LIN {X 0,Y 264.267,Z 962.971,A -85,B 0,C 180,E1 -27558.932,E2 -27558.932} C_VEL
LIN {X 0,Y 248.377,Z 979.382,A -85,B 0,C 180,E1 -27561.576,E2 -27561.576} C_VEL
LIN {X 0,Y 232.266,Z 994.174,A -85,B 0,C 180,E1 -27564.723,E2 -27564.723} C_VEL
LIN {X 0,Y 216.727,Z 1007.351,A -85,B 0,C 180,E1 -27568.372,E2 -27568.372} C_VEL
LIN {X 0,Y 201.146,Z 1019.293,A -85,B 0,C 180,E1 -27572.85,E2 -27572.85} C_VEL
LIN {X 0,Y 187.229,Z 1029.33,A -85,B 0,C 180,E1 -27577.891,E2 -27577.891} C_VEL
LIN {X 0,Y 173.48,Z 1038.583,A -85,B 0,C 180,E1 -27584.382,E2 -27584.382} C_VEL
LIN {X 0,Y 162.777,Z 1045.623,A -85,B 0,C 180,E1 -27591.272,E2 -27591.272} C_VEL
LIN {X 0,Y 153.415,Z 1051.791,A -85,B 0,C 180,E1 -27600.094,E2 -27600.094} C_VEL
LIN {X 0,Y 148.288,Z 1055.438,A -85,B 0,C 180,E1 -27607.815,E2 -27607.815} C_VEL
LIN {X 0,Y 145.02,Z 1058.302,A -85,B 0,C 180,E1 -27617.254,E2 -27617.254} C_VEL
LIN {X 0,Y 144.131,Z 1059.404,A -85,B 0,C 180,E1 -27625.225,E2 -27625.225} C_VEL
LIN {X 0,Y 144.059,Z 1059.565,A -85,B 0,C 180,E1 -27631.989,E2 -27631.989} C_VEL
LIN {X 0,Y 144.452,Z 1058.916,A -85,B 0,C 180,E1 -27639.161,E2 -27639.161} C_VEL
LIN {X 0,Y 146.018,Z 1057.309,A -85,B 0,C 180,E1 -27646.715,E2 -27646.715} C_VEL
LIN {X 0,Y 149.982,Z 1054.279,A -85,B 0,C 180,E1 -27655.257,E2 -27655.257} C_VEL
LIN {X 0,Y 157.615,Z 1049.051,A -85,B 0,C 180,E1 -27664.441,E2 -27664.441} C_VEL
LIN {X 0,Y 166.845,Z 1043.052,A -85,B 0,C 180,E1 -27671.699,E2 -27671.699} C_VEL
LIN {X 0,Y 180.107,Z 1034.277,A -85,B 0,C 180,E1 -27679.073,E2 -27679.073} C_VEL
LIN {X 0,Y 192.349,Z 1025.823,A -85,B 0,C 180,E1 -27684.188,E2 -27684.188} C_VEL
LIN {X 0,Y 208.78,Z 1013.706,A -85,B 0,C 180,E1 -27689.548,E2 -27689.548} C_VEL
LIN {X 0,Y 222.856,Z 1002.432,A -85,B 0,C 180,E1 -27693.234,E2 -27693.234} C_VEL
LIN {X 0,Y 239.33,Z 988.118,A -85,B 0,C 180,E1 -27696.8,E2 -27696.8} C_VEL
LIN {X 0,Y 254.068,Z 973.895,A -85,B 0,C 180,E1 -27699.497,E2 -27699.497} C_VEL
LIN {X 0,Y 269.736,Z 957.383,A -85,B 0,C 180,E1 -27701.958,E2 -27701.958} C_VEL
LIN {X 0,Y 284.481,Z 939.789,A -85,B 0,C 180,E1 -27703.988,E2 -27703.988} C_VEL
LIN {X 0,Y 298.698,Z 921.024,A -85,B 0,C 180,E1 -27705.72,E2 -27705.72} C_VEL
LIN {X 0,Y 311.756,Z 901.235,A -85,B 0,C 180,E1 -27707.166,E2 -27707.166} C_VEL
LIN {X 0,Y 323.633,Z 881.021,A -85,B 0,C 180,E1 -27708.35,E2 -27708.35} C_VEL
LIN {X 0,Y 334.691,Z 859.013,A -85,B 0,C 180,E1 -27709.386,E2 -27709.386} C_VEL
LIN {X 0,Y 343.522,Z 838.703,A -85,B 0,C 180,E1 -27710.155,E2 -27710.155} C_VEL
LIN {X 0,Y 352.143,Z 814.942,A -85,B 0,C 180,E1 -27710.876,E2 -27710.876} C_VEL
LIN {X 0,Y 358.427,Z 793.654,A -85,B 0,C 180,E1 -27711.389,E2 -27711.389} C_VEL
LIN {X 0,Y 364.35,Z 767.82,A -85,B 0,C 180,E1 -27711.861,E2 -27711.861} C_VEL
LIN {X 0,Y 367.939,Z 745.502,A -85,B 0,C 180,E1 -27712.18,E2 -27712.18} C_VEL
LIN {X 0,Y 380.155,Z 638.893,A -85,B 0,C 180,E1 -27713.582,E2 -27713.582} C_VEL
LIN {X 0,Y 379.242,Z 636.279,A -85,B 0,C 180,E1 -27715.615,E2 -27715.615} C_VEL
LIN {X 0,Y 378.541,Z 633.63,A -85,B 0,C 180,E1 -27720,E2 -27720} C_VEL
LIN {X 0,Y 379.492,Z 636.936,A -85,B 0,C 180,E1 -27724.685,E2 -27724.685} C_VEL
LIN {X 0,Y 380.192,Z 639.051,A -85,B 0,C 180,E1 -27726.164,E2 -27726.164} C_VEL
LIN {X 0,Y 366.89,Z 754.069,A -85,B 0,C 180,E1 -27727.662,E2 -27727.662} C_VEL
LIN {X 0,Y 362.071,Z 780.264,A -85,B 0,C 180,E1 -27728.054,E2 -27728.054} C_VEL
LIN {X 0,Y 356.568,Z 802.149,A -85,B 0,C 180,E1 -27728.434,E2 -27728.434} C_VEL
LIN {X 0,Y 353.055,Z 813.807,A -85,B 0,C 180,E1 -27728.68,E2 -27728.68} C_VEL
LIN {X 0,Y 350.527,Z 821.162,A -85,B 0,C 180,E1 -27728.649,E2 -27728.649} C_VEL
LIN {X 0,Y 342.323,Z 840.671,A -85,B 0,C 180,E1 -27728.173,E2 -27728.173} C_VEL
LIN {X 0,Y 339.699,Z 846.579,A -85,B 0,C 180,E1 -27728.225,E2 -27728.225} C_VEL
LIN {X 0,Y 329.393,Z 869.145,A -85,B 0,C 180,E1 -27729.009,E2 -27729.009} C_VEL
LIN {X 0,Y 318.229,Z 889.834,A -85,B 0,C 180,E1 -27729.926,E2 -27729.926} C_VEL
LIN {X 0,Y 305.654,Z 910.454,A -85,B 0,C 180,E1 -27731.069,E2 -27731.069} C_VEL
LIN {X 0,Y 291.612,Z 930.378,A -85,B 0,C 180,E1 -27732.475,E2 -27732.475} C_VEL
LIN {X 0,Y 277.331,Z 948.589,A -85,B 0,C 180,E1 -27734.104,E2 -27734.104} C_VEL
LIN {X 0,Y 261.326,Z 966.611,A -85,B 0,C 180,E1 -27736.181,E2 -27736.181} C_VEL
LIN {X 0,Y 246.138,Z 982.117,A -85,B 0,C 180,E1 -27738.473,E2 -27738.473} C_VEL
LIN {X 0,Y 228.96,Z 997.86,A -85,B 0,C 180,E1 -27741.535,E2 -27741.535} C_VEL
LIN {X 0,Y 213.707,Z 1010.632,A -85,B 0,C 180,E1 -27744.812,E2 -27744.812} C_VEL
LIN {X 0,Y 196.327,Z 1023.93,A -85,B 0,C 180,E1 -27749.436,E2 -27749.436} C_VEL
LIN {X 0,Y 182.4,Z 1033.814,A -85,B 0,C 180,E1 -27754.13,E2 -27754.13} C_VEL
LIN {X 0,Y 166.948,Z 1044.167,A -85,B 0,C 180,E1 -27761.006,E2 -27761.006} C_VEL
LIN {X 0,Y 156.007,Z 1051.247,A -85,B 0,C 180,E1 -27767.703,E2 -27767.703} C_VEL
LIN {X 0,Y 145.908,Z 1057.948,A -85,B 0,C 180,E1 -27776.754,E2 -27776.754} C_VEL
LIN {X 0,Y 139.953,Z 1062.241,A -85,B 0,C 180,E1 -27785.519,E2 -27785.519} C_VEL
LIN {X 0,Y 136.886,Z 1065.116,A -85,B 0,C 180,E1 -27794.319,E2 -27794.319} C_VEL
LIN {X 0,Y 135.998,Z 1066.786,A -85,B 0,C 180,E1 -27803.668,E2 -27803.668} C_VEL
LIN {X 0,Y 136.048,Z 1067.121,A -85,B 0,C 180,E1 -27810.421,E2 -27810.421} C_VEL
LIN {X 0,Y 136.022,Z 1066.636,A -85,B 0,C 180,E1 -27817.603,E2 -27817.603} C_VEL
LIN {X 0,Y 137.072,Z 1064.849,A -85,B 0,C 180,E1 -27826.528,E2 -27826.528} C_VEL
LIN {X 0,Y 140.303,Z 1061.923,A -85,B 0,C 180,E1 -27835.165,E2 -27835.165} C_VEL
LIN {X 0,Y 147.301,Z 1056.96,A -85,B 0,C 180,E1 -27844.778,E2 -27844.778} C_VEL
LIN {X 0,Y 156.952,Z 1050.544,A -85,B 0,C 180,E1 -27852.973,E2 -27852.973} C_VEL
LIN {X 0,Y 169.249,Z 1042.625,A -85,B 0,C 180,E1 -27860.176,E2 -27860.176} C_VEL
LIN {X 0,Y 183.726,Z 1032.758,A -85,B 0,C 180,E1 -27866.373,E2 -27866.373} C_VEL
LIN {X 0,Y 199.243,Z 1021.702,A -85,B 0,C 180,E1 -27871.429,E2 -27871.429} C_VEL
LIN {X 0,Y 215.441,Z 1009.024,A -85,B 0,C 180,E1 -27875.603,E2 -27875.603} C_VEL
LIN {X 0,Y 230.594,Z 996.24,A -85,B 0,C 180,E1 -27878.791,E2 -27878.791} C_VEL
LIN {X 0,Y 247.424,Z 980.57,A -85,B 0,C 180,E1 -27881.746,E2 -27881.746} C_VEL
LIN {X 0,Y 261.312,Z 966.334,A -85,B 0,C 180,E1 -27883.828,E2 -27883.828} C_VEL
LIN {X 0,Y 277.317,Z 948.252,A -85,B 0,C 180,E1 -27885.906,E2 -27885.906} C_VEL
LIN {X 0,Y 291.424,Z 930.233,A -85,B 0,C 180,E1 -27887.517,E2 -27887.517} C_VEL
LIN {X 0,Y 305.178,Z 910.722,A -85,B 0,C 180,E1 -27888.897,E2 -27888.897} C_VEL
LIN {X 0,Y 317.749,Z 890.132,A -85,B 0,C 180,E1 -27890.045,E2 -27890.045} C_VEL
LIN {X 0,Y 328.563,Z 870.14,A -85,B 0,C 180,E1 -27890.939,E2 -27890.939} C_VEL
LIN {X 0,Y 338.982,Z 847.539,A -85,B 0,C 180,E1 -27891.736,E2 -27891.736} C_VEL
LIN {X 0,Y 347.083,Z 826.938,A -85,B 0,C 180,E1 -27892.309,E2 -27892.309} C_VEL
LIN {X 0,Y 355.377,Z 801.149,A -85,B 0,C 180,E1 -27892.854,E2 -27892.854} C_VEL
LIN {X 0,Y 360.895,Z 779.258,A -85,B 0,C 180,E1 -27893.213,E2 -27893.213} C_VEL
LIN {X 0,Y 365.786,Z 752.36,A -85,B 0,C 180,E1 -27893.598,E2 -27893.598} C_VEL
LIN {X 0,Y 378.338,Z 645.252,A -85,B 0,C 180,E1 -27894.959,E2 -27894.959} C_VEL
LIN {X 0,Y 377.845,Z 643.846,A -85,B 0,C 180,E1 -27896.207,E2 -27896.207} C_VEL
LIN {X 0,Y 377.267,Z 641.047,A -85,B 0,C 180,E1 -27900.304,E2 -27900.304} C_VEL
LIN {X 0,Y 378.12,Z 644.537,A -85,B 0,C 180,E1 -27904.93,E2 -27904.93} C_VEL
LIN {X 0,Y 378.282,Z 645.473,A -85,B 0,C 180,E1 -27905.413,E2 -27905.413} C_VEL
LIN {X 0,Y 365.783,Z 751.706,A -85,B 0,C 180,E1 -27906.758,E2 -27906.758} C_VEL
LIN {X 0,Y 360.96,Z 777.648,A -85,B 0,C 180,E1 -27907.144,E2 -27907.144} C_VEL
LIN {X 0,Y 355.511,Z 799.249,A -85,B 0,C 180,E1 -27907.55,E2 -27907.55} C_VEL
LIN {X 0,Y 347.486,Z 824.285,A -85,B 0,C 180,E1 -27908.168,E2 -27908.168} C_VEL
LIN {X 0,Y 339.282,Z 845.216,A -85,B 0,C 180,E1 -27908.831,E2 -27908.831} C_VEL
LIN {X 0,Y 328.693,Z 868.101,A -85,B 0,C 180,E1 -27909.732,E2 -27909.732} C_VEL
LIN {X 0,Y 318.082,Z 887.67,A -85,B 0,C 180,E1 -27910.688,E2 -27910.688} C_VEL
LIN {X 0,Y 305.545,Z 908.098,A -85,B 0,C 180,E1 -27911.911,E2 -27911.911} C_VEL
LIN {X 0,Y 291.891,Z 927.376,A -85,B 0,C 180,E1 -27913.38,E2 -27913.38} C_VEL
LIN {X 0,Y 277.553,Z 945.569,A -85,B 0,C 180,E1 -27915.101,E2 -27915.101} C_VEL
LIN {X 0,Y 262.605,Z 962.274,A -85,B 0,C 180,E1 -27917.119,E2 -27917.119} C_VEL
LIN {X 0,Y 248.018,Z 977.098,A -85,B 0,C 180,E1 -27919.374,E2 -27919.374} C_VEL
LIN {X 0,Y 230.582,Z 993.009,A -85,B 0,C 180,E1 -27922.536,E2 -27922.536} C_VEL
LIN {X 0,Y 216.255,Z 1004.884,A -85,B 0,C 180,E1 -27925.629,E2 -27925.629} C_VEL
LIN {X 0,Y 198.972,Z 1017.992,A -85,B 0,C 180,E1 -27930.192,E2 -27930.192} C_VEL
LIN {X 0,Y 185.069,Z 1027.645,A -85,B 0,C 180,E1 -27934.793,E2 -27934.793} C_VEL
LIN {X 0,Y 170.308,Z 1037.306,A -85,B 0,C 180,E1 -27941.114,E2 -27941.114} C_VEL
LIN {X 0,Y 158.413,Z 1044.613,A -85,B 0,C 180,E1 -27948.006,E2 -27948.006} C_VEL
LIN {X 0,Y 148.285,Z 1050.907,A -85,B 0,C 180,E1 -27956.432,E2 -27956.432} C_VEL
LIN {X 0,Y 141.455,Z 1055.193,A -85,B 0,C 180,E1 -27965.352,E2 -27965.352} C_VEL
LIN {X 0,Y 137.778,Z 1057.908,A -85,B 0,C 180,E1 -27973.992,E2 -27973.992} C_VEL
LIN {X 0,Y 136.239,Z 1059.536,A -85,B 0,C 180,E1 -27983.257,E2 -27983.257} C_VEL
LIN {X 0,Y 136.057,Z 1059.844,A -85,B 0,C 180,E1 -27990.843,E2 -27990.843} C_VEL
LIN {X 0,Y 136.415,Z 1059.26,A -85,B 0,C 180,E1 -27998.855,E2 -27998.855} C_VEL
LIN {X 0,Y 138.135,Z 1057.635,A -85,B 0,C 180,E1 -28007.265,E2 -28007.265} C_VEL
LIN {X 0,Y 142.135,Z 1054.805,A -85,B 0,C 180,E1 -28015.859,E2 -28015.859} C_VEL
LIN {X 0,Y 150.472,Z 1049.553,A -85,B 0,C 180,E1 -28025.787,E2 -28025.787} C_VEL
LIN {X 0,Y 159.802,Z 1043.863,A -85,B 0,C 180,E1 -28033.002,E2 -28033.002} C_VEL
LIN {X 0,Y 173.564,Z 1035.328,A -85,B 0,C 180,E1 -28040.531,E2 -28040.531} C_VEL
LIN {X 0,Y 186.98,Z 1026.493,A -85,B 0,C 180,E1 -28045.984,E2 -28045.984} C_VEL
LIN {X 0,Y 203.26,Z 1015.054,A -85,B 0,C 180,E1 -28051.12,E2 -28051.12} C_VEL
LIN {X 0,Y 218.5,Z 1003.277,A -85,B 0,C 180,E1 -28054.97,E2 -28054.97} C_VEL
LIN {X 0,Y 234.581,Z 989.845,A -85,B 0,C 180,E1 -28058.313,E2 -28058.313} C_VEL
LIN {X 0,Y 250.84,Z 974.588,A -85,B 0,C 180,E1 -28061.163,E2 -28061.163} C_VEL
LIN {X 0,Y 266.01,Z 958.994,A -85,B 0,C 180,E1 -28063.437,E2 -28063.437} C_VEL
LIN {X 0,Y 281.477,Z 941.075,A -85,B 0,C 180,E1 -28065.467,E2 -28065.467} C_VEL
LIN {X 0,Y 294.529,Z 924.26,A -85,B 0,C 180,E1 -28066.99,E2 -28066.99} C_VEL
LIN {X 0,Y 308.68,Z 903.638,A -85,B 0,C 180,E1 -28068.485,E2 -28068.485} C_VEL
LIN {X 0,Y 319.891,Z 885.068,A -85,B 0,C 180,E1 -28069.555,E2 -28069.555} C_VEL
LIN {X 0,Y 331.432,Z 863.224,A -85,B 0,C 180,E1 -28070.582,E2 -28070.582} C_VEL
LIN {X 0,Y 340.824,Z 842.289,A -85,B 0,C 180,E1 -28071.368,E2 -28071.368} C_VEL
LIN {X 0,Y 349.564,Z 819.498,A -85,B 0,C 180,E1 -28072.06,E2 -28072.06} C_VEL
LIN {X 0,Y 356.719,Z 796.023,A -85,B 0,C 180,E1 -28072.615,E2 -28072.615} C_VEL
LIN {X 0,Y 362.622,Z 771.737,A -85,B 0,C 180,E1 -28073.055,E2 -28073.055} C_VEL
LIN {X 0,Y 366.721,Z 747.257,A -85,B 0,C 180,E1 -28073.397,E2 -28073.397} C_VEL
LIN {X 0,Y 378.603,Z 645.5,A -85,B 0,C 180,E1 -28074.696,E2 -28074.696} C_VEL
LIN {X 0,Y 378.146,Z 644.074,A -85,B 0,C 180,E1 -28075.906,E2 -28075.906} C_VEL
LIN {X 0,Y 377.562,Z 641.607,A -85,B 0,C 180,E1 -28080,E2 -28080} C_VEL
LIN {X 0,Y 378.441,Z 644.845,A -85,B 0,C 180,E1 -28084.546,E2 -28084.546} C_VEL
LIN {X 0,Y 378.613,Z 645.771,A -85,B 0,C 180,E1 -28085.044,E2 -28085.044} C_VEL
LIN {X 0,Y 365.885,Z 754.02,A -85,B 0,C 180,E1 -28086.417,E2 -28086.417} C_VEL
LIN {X 0,Y 361.033,Z 780.062,A -85,B 0,C 180,E1 -28086.792,E2 -28086.792} C_VEL
LIN {X 0,Y 355.448,Z 802.054,A -85,B 0,C 180,E1 -28087.154,E2 -28087.154} C_VEL
LIN {X 0,Y 347.573,Z 826.478,A -85,B 0,C 180,E1 -28087.671,E2 -28087.671} C_VEL
LIN {X 0,Y 339.699,Z 846.579,A -85,B 0,C 180,E1 -28088.225,E2 -28088.225} C_VEL
LIN {X 0,Y 336.5,Z 853.766,A -85,B 0,C 180,E1 -28088.278,E2 -28088.278} C_VEL
LIN {X 0,Y 327.075,Z 871.41,A -85,B 0,C 180,E1 -28087.878,E2 -28087.878} C_VEL
LIN {X 0,Y 323.395,Z 878.079,A -85,B 0,C 180,E1 -28087.97,E2 -28087.97} C_VEL
LIN {X 0,Y 309.842,Z 901.381,A -85,B 0,C 180,E1 -28089.071,E2 -28089.071} C_VEL
LIN {X 0,Y 297.638,Z 919.683,A -85,B 0,C 180,E1 -28090.162,E2 -28090.162} C_VEL
LIN {X 0,Y 281.872,Z 940.552,A -85,B 0,C 180,E1 -28091.745,E2 -28091.745} C_VEL
LIN {X 0,Y 268.172,Z 956.644,A -85,B 0,C 180,E1 -28093.307,E2 -28093.307} C_VEL
LIN {X 0,Y 252.011,Z 973.807,A -85,B 0,C 180,E1 -28095.417,E2 -28095.417} C_VEL
LIN {X 0,Y 236.296,Z 988.661,A -85,B 0,C 180,E1 -28097.807,E2 -28097.807} C_VEL
LIN {X 0,Y 219.884,Z 1002.877,A -85,B 0,C 180,E1 -28100.775,E2 -28100.775} C_VEL
LIN {X 0,Y 202.401,Z 1016.446,A -85,B 0,C 180,E1 -28104.634,E2 -28104.634} C_VEL
LIN {X 0,Y 186.443,Z 1027.891,A -85,B 0,C 180,E1 -28109.053,E2 -28109.053} C_VEL
LIN {X 0,Y 170.442,Z 1038.405,A -85,B 0,C 180,E1 -28114.784,E2 -28114.784} C_VEL
LIN {X 0,Y 157.522,Z 1046.472,A -85,B 0,C 180,E1 -28120.942,E2 -28120.942} C_VEL
LIN {X 0,Y 144.759,Z 1054.201,A -85,B 0,C 180,E1 -28129.512,E2 -28129.512} C_VEL
LIN {X 0,Y 136.669,Z 1059.222,A -85,B 0,C 180,E1 -28137.718,E2 -28137.718} C_VEL
LIN {X 0,Y 130.717,Z 1063.469,A -85,B 0,C 180,E1 -28147.987,E2 -28147.987} C_VEL
LIN {X 0,Y 128.303,Z 1065.79,A -85,B 0,C 180,E1 -28157.853,E2 -28157.853} C_VEL
LIN {X 0,Y 128.002,Z 1066.673,A -85,B 0,C 180,E1 -28165.07,E2 -28165.07} C_VEL
LIN {X 0,Y 128.037,Z 1066.847,A -85,B 0,C 180,E1 -28171.611,E2 -28171.611} C_VEL
LIN {X 0,Y 128.061,Z 1066.277,A -85,B 0,C 180,E1 -28178.984,E2 -28178.984} C_VEL
LIN {X 0,Y 129.395,Z 1064.512,A -85,B 0,C 180,E1 -28188.004,E2 -28188.004} C_VEL
LIN {X 0,Y 133.243,Z 1061.482,A -85,B 0,C 180,E1 -28197.242,E2 -28197.242} C_VEL
LIN {X 0,Y 141.776,Z 1055.963,A -85,B 0,C 180,E1 -28207.848,E2 -28207.848} C_VEL
LIN {X 0,Y 152.078,Z 1049.679,A -85,B 0,C 180,E1 -28215.818,E2 -28215.818} C_VEL
LIN {X 0,Y 166.561,Z 1040.767,A -85,B 0,C 180,E1 -28223.554,E2 -28223.554} C_VEL
LIN {X 0,Y 180.674,Z 1031.602,A -85,B 0,C 180,E1 -28229.07,E2 -28229.07} C_VEL
LIN {X 0,Y 197.714,Z 1019.773,A -85,B 0,C 180,E1 -28234.182,E2 -28234.182} C_VEL
LIN {X 0,Y 213.604,Z 1007.659,A -85,B 0,C 180,E1 -28237.948,E2 -28237.948} C_VEL
LIN {X 0,Y 231.168,Z 993.076,A -85,B 0,C 180,E1 -28241.332,E2 -28241.332} C_VEL
LIN {X 0,Y 246.727,Z 978.641,A -85,B 0,C 180,E1 -28243.835,E2 -28243.835} C_VEL
LIN {X 0,Y 262.742,Z 962.378,A -85,B 0,C 180,E1 -28246.03,E2 -28246.03} C_VEL
LIN {X 0,Y 278.183,Z 944.676,A -85,B 0,C 180,E1 -28247.867,E2 -28247.867} C_VEL
LIN {X 0,Y 291.565,Z 927.644,A -85,B 0,C 180,E1 -28249.27,E2 -28249.27} C_VEL
LIN {X 0,Y 306.532,Z 906.072,A -85,B 0,C 180,E1 -28250.657,E2 -28250.657} C_VEL
LIN {X 0,Y 317.663,Z 887.817,A -85,B 0,C 180,E1 -28251.592,E2 -28251.592} C_VEL
LIN {X 0,Y 329.774,Z 865.097,A -85,B 0,C 180,E1 -28252.513,E2 -28252.513} C_VEL
LIN {X 0,Y 339.026,Z 844.701,A -85,B 0,C 180,E1 -28253.163,E2 -28253.163} C_VEL
LIN {X 0,Y 348.03,Z 821.467,A -85,B 0,C 180,E1 -28253.749,E2 -28253.749} C_VEL
LIN {X 0,Y 355.282,Z 797.991,A -85,B 0,C 180,E1 -28254.193,E2 -28254.193} C_VEL
LIN {X 0,Y 361.272,Z 773.573,A -85,B 0,C 180,E1 -28254.563,E2 -28254.563} C_VEL
LIN {X 0,Y 365.395,Z 749.119,A -85,B 0,C 180,E1 -28254.89,E2 -28254.89} C_VEL
LIN {X 0,Y 376.897,Z 651.874,A -85,B 0,C 180,E1 -28256.121,E2 -28256.121} C_VEL
LIN {X 0,Y 376.286,Z 649.042,A -85,B 0,C 180,E1 -28260.305,E2 -28260.305} C_VEL
LIN {X 0,Y 376.874,Z 651.979,A -85,B 0,C 180,E1 -28264.279,E2 -28264.279} C_VEL
LIN {X 0,Y 364.904,Z 752.116,A -85,B 0,C 180,E1 -28265.512,E2 -28265.512} C_VEL
LIN {X 0,Y 360.049,Z 777.886,A -85,B 0,C 180,E1 -28265.88,E2 -28265.88} C_VEL
LIN {X 0,Y 354.531,Z 799.534,A -85,B 0,C 180,E1 -28266.268,E2 -28266.268} C_VEL
LIN {X 0,Y 346.437,Z 824.507,A -85,B 0,C 180,E1 -28266.854,E2 -28266.854} C_VEL
LIN {X 0,Y 338.312,Z 845.035,A -85,B 0,C 180,E1 -28267.472,E2 -28267.472} C_VEL
LIN {X 0,Y 327.901,Z 867.426,A -85,B 0,C 180,E1 -28268.304,E2 -28268.304} C_VEL
LIN {X 0,Y 317.061,Z 887.243,A -85,B 0,C 180,E1 -28269.22,E2 -28269.22} C_VEL
LIN {X 0,Y 304.443,Z 907.627,A -85,B 0,C 180,E1 -28270.374,E2 -28270.374} C_VEL
LIN {X 0,Y 290.581,Z 926.992,A -85,B 0,C 180,E1 -28271.773,E2 -28271.773} C_VEL
LIN {X 0,Y 276.451,Z 944.688,A -85,B 0,C 180,E1 -28273.36,E2 -28273.36} C_VEL
LIN {X 0,Y 260.324,Z 962.495,A -85,B 0,C 180,E1 -28275.405,E2 -28275.405} C_VEL
LIN {X 0,Y 245.431,Z 977.318,A -85,B 0,C 180,E1 -28277.576,E2 -28277.576} C_VEL
LIN {X 0,Y 227.57,Z 993.23,A -85,B 0,C 180,E1 -28280.631,E2 -28280.631} C_VEL
LIN {X 0,Y 212.836,Z 1005.105,A -85,B 0,C 180,E1 -28283.638,E2 -28283.638} C_VEL
LIN {X 0,Y 194.97,Z 1018.213,A -85,B 0,C 180,E1 -28288.105,E2 -28288.105} C_VEL
LIN {X 0,Y 180.504,Z 1027.866,A -85,B 0,C 180,E1 -28292.649,E2 -28292.649} C_VEL
LIN {X 0,Y 165.431,Z 1037.293,A -85,B 0,C 180,E1 -28298.768,E2 -28298.768} C_VEL
LIN {X 0,Y 152.41,Z 1044.833,A -85,B 0,C 180,E1 -28305.94,E2 -28305.94} C_VEL
LIN {X 0,Y 141.535,Z 1051.126,A -85,B 0,C 180,E1 -28314.599,E2 -28314.599} C_VEL
LIN {X 0,Y 133.837,Z 1055.565,A -85,B 0,C 180,E1 -28324.322,E2 -28324.322} C_VEL
LIN {X 0,Y 129.755,Z 1058.344,A -85,B 0,C 180,E1 -28333.894,E2 -28333.894} C_VEL
LIN {X 0,Y 128.208,Z 1059.791,A -85,B 0,C 180,E1 -28343.732,E2 -28343.732} C_VEL
LIN {X 0,Y 128.062,Z 1060.035,A -85,B 0,C 180,E1 -28351.343,E2 -28351.343} C_VEL
LIN {X 0,Y 128.471,Z 1059.475,A -85,B 0,C 180,E1 -28359.407,E2 -28359.407} C_VEL
LIN {X 0,Y 130.413,Z 1057.851,A -85,B 0,C 180,E1 -28368.322,E2 -28368.322} C_VEL
LIN {X 0,Y 134.841,Z 1055.022,A -85,B 0,C 180,E1 -28377.371,E2 -28377.371} C_VEL
LIN {X 0,Y 143.899,Z 1049.771,A -85,B 0,C 180,E1 -28387.696,E2 -28387.696} C_VEL
LIN {X 0,Y 153.895,Z 1044.081,A -85,B 0,C 180,E1 -28395.089,E2 -28395.089} C_VEL
LIN {X 0,Y 167.826,Z 1035.944,A -85,B 0,C 180,E1 -28402.411,E2 -28402.411} C_VEL
LIN {X 0,Y 181.805,Z 1027.162,A -85,B 0,C 180,E1 -28407.884,E2 -28407.884} C_VEL
LIN {X 0,Y 197.9,Z 1016.396,A -85,B 0,C 180,E1 -28412.779,E2 -28412.779} C_VEL
LIN {X 0,Y 214.351,Z 1004.121,A -85,B 0,C 180,E1 -28416.774,E2 -28416.774} C_VEL
LIN {X 0,Y 230.838,Z 990.757,A -85,B 0,C 180,E1 -28420.044,E2 -28420.044} C_VEL
LIN {X 0,Y 247.08,Z 976,A -85,B 0,C 180,E1 -28422.756,E2 -28422.756} C_VEL
LIN {X 0,Y 261.13,Z 961.963,A -85,B 0,C 180,E1 -28424.781,E2 -28424.781} C_VEL
LIN {X 0,Y 278.07,Z 943.085,A -85,B 0,C 180,E1 -28426.907,E2 -28426.907} C_VEL
LIN {X 0,Y 291.429,Z 926.286,A -85,B 0,C 180,E1 -28428.392,E2 -28428.392} C_VEL
LIN {X 0,Y 305.772,Z 906.042,A -85,B 0,C 180,E1 -28429.83,E2 -28429.83} C_VEL
LIN {X 0,Y 317.471,Z 887.094,A -85,B 0,C 180,E1 -28430.89,E2 -28430.89} C_VEL
LIN {X 0,Y 328.953,Z 866.044,A -85,B 0,C 180,E1 -28431.855,E2 -28431.855} C_VEL
LIN {X 0,Y 338.758,Z 844.749,A -85,B 0,C 180,E1 -28432.635,E2 -28432.635} C_VEL
LIN {X 0,Y 346.867,Z 824.239,A -85,B 0,C 180,E1 -28433.249,E2 -28433.249} C_VEL
LIN {X 0,Y 355.048,Z 798.859,A -85,B 0,C 180,E1 -28433.842,E2 -28433.842} C_VEL
LIN {X 0,Y 360.569,Z 777.071,A -85,B 0,C 180,E1 -28434.23,E2 -28434.23} C_VEL
LIN {X 0,Y 365.485,Z 750.335,A -85,B 0,C 180,E1 -28434.606,E2 -28434.606} C_VEL
LIN {X 0,Y 377.199,Z 652.091,A -85,B 0,C 180,E1 -28435.819,E2 -28435.819} C_VEL
LIN {X 0,Y 376.582,Z 649.582,A -85,B 0,C 180,E1 -28440,E2 -28440} C_VEL
LIN {X 0,Y 377.201,Z 652.309,A -85,B 0,C 180,E1 -28443.913,E2 -28443.913} C_VEL
LIN {X 0,Y 365.076,Z 753.823,A -85,B 0,C 180,E1 -28445.165,E2 -28445.165} C_VEL
LIN {X 0,Y 360.144,Z 779.979,A -85,B 0,C 180,E1 -28445.525,E2 -28445.525} C_VEL
LIN {X 0,Y 354.506,Z 801.959,A -85,B 0,C 180,E1 -28445.867,E2 -28445.867} C_VEL
LIN {X 0,Y 346.59,Z 826.271,A -85,B 0,C 180,E1 -28446.351,E2 -28446.351} C_VEL
LIN {X 0,Y 338.24,Z 847.311,A -85,B 0,C 180,E1 -28446.901,E2 -28446.901} C_VEL
LIN {X 0,Y 327.875,Z 869.594,A -85,B 0,C 180,E1 -28447.64,E2 -28447.64} C_VEL
LIN {X 0,Y 323.395,Z 878.079,A -85,B 0,C 180,E1 -28447.97,E2 -28447.97} C_VEL
LIN {X 0,Y 319.555,Z 884.853,A -85,B 0,C 180,E1 -28448.078,E2 -28448.078} C_VEL
LIN {X 0,Y 308.524,Z 901.631,A -85,B 0,C 180,E1 -28447.786,E2 -28447.786} C_VEL
LIN {X 0,Y 304.263,Z 907.989,A -85,B 0,C 180,E1 -28447.938,E2 -28447.938} C_VEL
LIN {X 0,Y 289.417,Z 928.793,A -85,B 0,C 180,E1 -28449.227,E2 -28449.227} C_VEL
LIN {X 0,Y 275.661,Z 945.924,A -85,B 0,C 180,E1 -28450.584,E2 -28450.584} C_VEL
LIN {X 0,Y 258.148,Z 965.245,A -85,B 0,C 180,E1 -28452.557,E2 -28452.557} C_VEL
LIN {X 0,Y 243.077,Z 980.109,A -85,B 0,C 180,E1 -28454.532,E2 -28454.532} C_VEL
LIN {X 0,Y 224.294,Z 996.716,A -85,B 0,C 180,E1 -28457.446,E2 -28457.446} C_VEL
LIN {X 0,Y 208.975,Z 1008.909,A -85,B 0,C 180,E1 -28460.313,E2 -28460.313} C_VEL
LIN {X 0,Y 191.086,Z 1021.923,A -85,B 0,C 180,E1 -28464.427,E2 -28464.427} C_VEL
LIN {X 0,Y 175.092,Z 1032.441,A -85,B 0,C 180,E1 -28469.105,E2 -28469.105} C_VEL
LIN {X 0,Y 159.14,Z 1042.284,A -85,B 0,C 180,E1 -28475.234,E2 -28475.234} C_VEL
LIN {X 0,Y 145.278,Z 1050.186,A -85,B 0,C 180,E1 -28482.571,E2 -28482.571} C_VEL
LIN {X 0,Y 133.636,Z 1056.854,A -85,B 0,C 180,E1 -28491.609,E2 -28491.609} C_VEL
LIN {X 0,Y 125.456,Z 1061.638,A -85,B 0,C 180,E1 -28501.95,E2 -28501.95} C_VEL
LIN {X 0,Y 121.399,Z 1064.563,A -85,B 0,C 180,E1 -28511.761,E2 -28511.761} C_VEL
LIN {X 0,Y 120.022,Z 1066.338,A -85,B 0,C 180,E1 -28522.472,E2 -28522.472} C_VEL
LIN {X 0,Y 120.061,Z 1066.713,A -85,B 0,C 180,E1 -28530,E2 -28530} C_VEL
LIN {X 0,Y 120.026,Z 1066.324,A -85,B 0,C 180,E1 -28537.659,E2 -28537.659} C_VEL
LIN {X 0,Y 121.399,Z 1064.531,A -85,B 0,C 180,E1 -28548.239,E2 -28548.239} C_VEL
LIN {X 0,Y 125.452,Z 1061.594,A -85,B 0,C 180,E1 -28558.05,E2 -28558.05} C_VEL
LIN {X 0,Y 133.632,Z 1056.786,A -85,B 0,C 180,E1 -28568.392,E2 -28568.392} C_VEL
LIN {X 0,Y 145.272,Z 1050.1,A -85,B 0,C 180,E1 -28577.431,E2 -28577.431} C_VEL
LIN {X 0,Y 159.132,Z 1042.18,A -85,B 0,C 180,E1 -28584.769,E2 -28584.769} C_VEL
LIN {X 0,Y 175.084,Z 1032.312,A -85,B 0,C 180,E1 -28590.899,E2 -28590.899} C_VEL
LIN {X 0,Y 191.867,Z 1021.256,A -85,B 0,C 180,E1 -28595.781,E2 -28595.781} C_VEL
LIN {X 0,Y 208.964,Z 1008.723,A -85,B 0,C 180,E1 -28599.694,E2 -28599.694} C_VEL
LIN {X 0,Y 225.151,Z 995.796,A -85,B 0,C 180,E1 -28602.709,E2 -28602.709} C_VEL
LIN {X 0,Y 242.94,Z 979.967,A -85,B 0,C 180,E1 -28605.459,E2 -28605.459} C_VEL
LIN {X 0,Y 258.137,Z 964.957,A -85,B 0,C 180,E1 -28607.452,E2 -28607.452} C_VEL
LIN {X 0,Y 275.65,Z 945.572,A -85,B 0,C 180,E1 -28609.426,E2 -28609.426} C_VEL
LIN {X 0,Y 289.23,Z 928.628,A -85,B 0,C 180,E1 -28610.767,E2 -28610.767} C_VEL
LIN {X 0,Y 304.104,Z 907.734,A -85,B 0,C 180,E1 -28612.062,E2 -28612.062} C_VEL
LIN {X 0,Y 315.827,Z 888.874,A -85,B 0,C 180,E1 -28612.988,E2 -28612.988} C_VEL
LIN {X 0,Y 327.372,Z 867.881,A -85,B 0,C 180,E1 -28613.809,E2 -28613.809} C_VEL
LIN {X 0,Y 337.527,Z 845.96,A -85,B 0,C 180,E1 -28614.481,E2 -28614.481} C_VEL
LIN {X 0,Y 345.784,Z 825.204,A -85,B 0,C 180,E1 -28614.986,E2 -28614.986} C_VEL
LIN {X 0,Y 353.859,Z 800.264,A -85,B 0,C 180,E1 -28615.446,E2 -28615.446} C_VEL
LIN {X 0,Y 359.472,Z 778.283,A -85,B 0,C 180,E1 -28615.765,E2 -28615.765} C_VEL
LIN {X 0,Y 364.36,Z 751.781,A -85,B 0,C 180,E1 -28616.112,E2 -28616.112} C_VEL
LIN {X 0,Y 375.552,Z 659.084,A -85,B 0,C 180,E1 -28617.253,E2 -28617.253} C_VEL
LIN {X 0,Y 375.304,Z 657.034,A -85,B 0,C 180,E1 -28620.305,E2 -28620.305} C_VEL
LIN {X 0,Y 375.524,Z 659.258,A -85,B 0,C 180,E1 -28623.147,E2 -28623.147} C_VEL
LIN {X 0,Y 364.208,Z 752.452,A -85,B 0,C 180,E1 -28624.26,E2 -28624.26} C_VEL
LIN {X 0,Y 359.315,Z 778.125,A -85,B 0,C 180,E1 -28624.61,E2 -28624.61} C_VEL
LIN {X 0,Y 353.728,Z 799.821,A -85,B 0,C 180,E1 -28624.979,E2 -28624.979} C_VEL
LIN {X 0,Y 345.572,Z 824.729,A -85,B 0,C 180,E1 -28625.534,E2 -28625.534} C_VEL
LIN {X 0,Y 337.247,Z 845.523,A -85,B 0,C 180,E1 -28626.127,E2 -28626.127} C_VEL
LIN {X 0,Y 326.357,Z 868.542,A -85,B 0,C 180,E1 -28626.943,E2 -28626.943} C_VEL
LIN {X 0,Y 315.868,Z 887.464,A -85,B 0,C 180,E1 -28627.775,E2 -28627.775} C_VEL
LIN {X 0,Y 303.091,Z 907.847,A -85,B 0,C 180,E1 -28628.87,E2 -28628.87} C_VEL
LIN {X 0,Y 289.036,Z 927.212,A -85,B 0,C 180,E1 -28630.2,E2 -28630.2} C_VEL
LIN {X 0,Y 274.688,Z 944.908,A -85,B 0,C 180,E1 -28631.711,E2 -28631.711} C_VEL
LIN {X 0,Y 258.28,Z 962.715,A -85,B 0,C 180,E1 -28633.663,E2 -28633.663} C_VEL
LIN {X 0,Y 242.969,Z 977.654,A -85,B 0,C 180,E1 -28635.76,E2 -28635.76} C_VEL
LIN {X 0,Y 224.817,Z 993.451,A -85,B 0,C 180,E1 -28638.679,E2 -28638.679} C_VEL
LIN {X 0,Y 209.683,Z 1005.326,A -85,B 0,C 180,E1 -28641.586,E2 -28641.586} C_VEL
LIN {X 0,Y 191.238,Z 1018.434,A -85,B 0,C 180,E1 -28645.934,E2 -28645.934} C_VEL
LIN {X 0,Y 176.205,Z 1028.087,A -85,B 0,C 180,E1 -28650.398,E2 -28650.398} C_VEL
LIN {X 0,Y 160.412,Z 1037.514,A -85,B 0,C 180,E1 -28656.478,E2 -28656.478} C_VEL
LIN {X 0,Y 146.621,Z 1045.053,A -85,B 0,C 180,E1 -28663.708,E2 -28663.708} C_VEL
LIN {X 0,Y 134.942,Z 1051.345,A -85,B 0,C 180,E1 -28672.584,E2 -28672.584} C_VEL
LIN {X 0,Y 126.541,Z 1055.783,A -85,B 0,C 180,E1 -28682.723,E2 -28682.723} C_VEL
LIN {X 0,Y 121.997,Z 1058.56,A -85,B 0,C 180,E1 -28692.839,E2 -28692.839} C_VEL
LIN {X 0,Y 120.234,Z 1060.005,A -85,B 0,C 180,E1 -28703.314,E2 -28703.314} C_VEL
LIN {X 0,Y 120.065,Z 1060.249,A -85,B 0,C 180,E1 -28711.432,E2 -28711.432} C_VEL
LIN {X 0,Y 120.533,Z 1059.689,A -85,B 0,C 180,E1 -28720.033,E2 -28720.033} C_VEL
LIN {X 0,Y 122.739,Z 1058.067,A -85,B 0,C 180,E1 -28729.513,E2 -28729.513} C_VEL
LIN {X 0,Y 127.65,Z 1055.239,A -85,B 0,C 180,E1 -28739.056,E2 -28739.056} C_VEL
LIN {X 0,Y 137.5,Z 1049.989,A -85,B 0,C 180,E1 -28749.787,E2 -28749.787} C_VEL
LIN {X 0,Y 148.209,Z 1044.3,A -85,B 0,C 180,E1 -28757.339,E2 -28757.339} C_VEL
LIN {X 0,Y 163.604,Z 1035.765,A -85,B 0,C 180,E1 -28764.982,E2 -28764.982} C_VEL
LIN {X 0,Y 178.3,Z 1026.929,A -85,B 0,C 180,E1 -28770.369,E2 -28770.369} C_VEL
LIN {X 0,Y 195.854,Z 1015.489,A -85,B 0,C 180,E1 -28775.332,E2 -28775.332} C_VEL
LIN {X 0,Y 212.253,Z 1003.582,A -85,B 0,C 180,E1 -28779.021,E2 -28779.021} C_VEL
LIN {X 0,Y 229.902,Z 989.529,A -85,B 0,C 180,E1 -28782.265,E2 -28782.265} C_VEL
LIN {X 0,Y 245.672,Z 975.378,A -85,B 0,C 180,E1 -28784.709,E2 -28784.709} C_VEL
LIN {X 0,Y 260.925,Z 960.341,A -85,B 0,C 180,E1 -28786.744,E2 -28786.744} C_VEL
LIN {X 0,Y 277.385,Z 942.053,A -85,B 0,C 180,E1 -28788.661,E2 -28788.661} C_VEL
LIN {X 0,Y 290.841,Z 925.289,A -85,B 0,C 180,E1 -28790.053,E2 -28790.053} C_VEL
LIN {X 0,Y 305.656,Z 904.382,A -85,B 0,C 180,E1 -28791.436,E2 -28791.436} C_VEL
LIN {X 0,Y 317.196,Z 885.77,A -85,B 0,C 180,E1 -28792.408,E2 -28792.408} C_VEL
LIN {X 0,Y 329.18,Z 863.641,A -85,B 0,C 180,E1 -28793.349,E2 -28793.349} C_VEL
LIN {X 0,Y 338.785,Z 842.704,A -85,B 0,C 180,E1 -28794.056,E2 -28794.056} C_VEL
LIN {X 0,Y 347.711,Z 819.908,A -85,B 0,C 180,E1 -28794.679,E2 -28794.679} C_VEL
LIN {X 0,Y 355.029,Z 796.382,A -85,B 0,C 180,E1 -28795.182,E2 -28795.182} C_VEL
LIN {X 0,Y 361.055,Z 772.033,A -85,B 0,C 180,E1 -28795.579,E2 -28795.579} C_VEL
LIN {X 0,Y 365.226,Z 747.641,A -85,B 0,C 180,E1 -28795.893,E2 -28795.893} C_VEL
LIN {X 0,Y 375.855,Z 659.371,A -85,B 0,C 180,E1 -28796.95,E2 -28796.95} C_VEL
LIN {X 0,Y 375.603,Z 657.559,A -85,B 0,C 180,E1 -28800,E2 -28800} C_VEL
LIN {X 0,Y 375.852,Z 659.564,A -85,B 0,C 180,E1 -28802.781,E2 -28802.781} C_VEL
LIN {X 0,Y 364.403,Z 753.898,A -85,B 0,C 180,E1 -28803.91,E2 -28803.91} C_VEL
LIN {X 0,Y 359.455,Z 779.8,A -85,B 0,C 180,E1 -28804.251,E2 -28804.251} C_VEL
LIN {X 0,Y 353.745,Z 801.864,A -85,B 0,C 180,E1 -28804.574,E2 -28804.574} C_VEL
LIN {X 0,Y 345.792,Z 826.065,A -85,B 0,C 180,E1 -28805.026,E2 -28805.026} C_VEL
LIN {X 0,Y 337.535,Z 846.709,A -85,B 0,C 180,E1 -28805.531,E2 -28805.531} C_VEL
LIN {X 0,Y 326.898,Z 869.384,A -85,B 0,C 180,E1 -28806.235,E2 -28806.235} C_VEL
LIN {X 0,Y 315.837,Z 889.411,A -85,B 0,C 180,E1 -28807.025,E2 -28807.025} C_VEL
LIN {X 0,Y 304.263,Z 907.989,A -85,B 0,C 180,E1 -28807.938,E2 -28807.938} C_VEL
LIN {X 0,Y 299.852,Z 914.346,A -85,B 0,C 180,E1 -28808.104,E2 -28808.104} C_VEL
LIN {X 0,Y 287.262,Z 930.021,A -85,B 0,C 180,E1 -28807.921,E2 -28807.921} C_VEL
LIN {X 0,Y 282.464,Z 935.989,A -85,B 0,C 180,E1 -28808.139,E2 -28808.139} C_VEL
LIN {X 0,Y 266.752,Z 954.171,A -85,B 0,C 180,E1 -28809.657,E2 -28809.657} C_VEL
LIN {X 0,Y 251.859,Z 969.696,A -85,B 0,C 180,E1 -28811.303,E2 -28811.303} C_VEL
LIN {X 0,Y 233.588,Z 986.67,A -85,B 0,C 180,E1 -28813.666,E2 -28813.666} C_VEL
LIN {X 0,Y 217.547,Z 1000.039,A -85,B 0,C 180,E1 -28816.135,E2 -28816.135} C_VEL
LIN {X 0,Y 197.755,Z 1014.846,A -85,B 0,C 180,E1 -28819.871,E2 -28819.871} C_VEL
LIN {X 0,Y 181.603,Z 1025.724,A -85,B 0,C 180,E1 -28823.699,E2 -28823.699} C_VEL
LIN {X 0,Y 163.001,Z 1037.139,A -85,B 0,C 180,E1 -28829.417,E2 -28829.417} C_VEL
LIN {X 0,Y 148.479,Z 1045.31,A -85,B 0,C 180,E1 -28835.428,E2 -28835.428} C_VEL
LIN {X 0,Y 134.186,Z 1052.977,A -85,B 0,C 180,E1 -28843.714,E2 -28843.714} C_VEL
LIN {X 0,Y 123.432,Z 1058.569,A -85,B 0,C 180,E1 -28853.169,E2 -28853.169} C_VEL
LIN {X 0,Y 115.915,Z 1062.906,A -85,B 0,C 180,E1 -28864.449,E2 -28864.449} C_VEL
LIN {X 0,Y 112.495,Z 1065.358,A -85,B 0,C 180,E1 -28876.114,E2 -28876.114} C_VEL
LIN {X 0,Y 112.006,Z 1066.269,A -85,B 0,C 180,E1 -28884.878,E2 -28884.878} C_VEL
LIN {X 0,Y 112.04,Z 1066.424,A -85,B 0,C 180,E1 -28891.738,E2 -28891.738} C_VEL
LIN {X 0,Y 112.129,Z 1065.845,A -85,B 0,C 180,E1 -28900.273,E2 -28900.273} C_VEL
LIN {X 0,Y 113.984,Z 1064.075,A -85,B 0,C 180,E1 -28910.541,E2 -28910.541} C_VEL
LIN {X 0,Y 118.9,Z 1061.021,A -85,B 0,C 180,E1 -28920.933,E2 -28920.933} C_VEL
LIN {X 0,Y 129.111,Z 1055.519,A -85,B 0,C 180,E1 -28932.358,E2 -28932.358} C_VEL
LIN {X 0,Y 140.981,Z 1049.257,A -85,B 0,C 180,E1 -28940.63,E2 -28940.63} C_VEL
LIN {X 0,Y 157.27,Z 1040.322,A -85,B 0,C 180,E1 -28948.423,E2 -28948.423} C_VEL
LIN {X 0,Y 172.731,Z 1031.156,A -85,B 0,C 180,E1 -28953.798,E2 -28953.798} C_VEL
LIN {X 0,Y 191.083,Z 1019.327,A -85,B 0,C 180,E1 -28958.658,E2 -28958.658} C_VEL
LIN {X 0,Y 207.961,Z 1007.214,A -85,B 0,C 180,E1 -28962.174,E2 -28962.174} C_VEL
LIN {X 0,Y 226.401,Z 992.655,A -85,B 0,C 180,E1 -28965.285,E2 -28965.285} C_VEL
LIN {X 0,Y 242.663,Z 978.197,A -85,B 0,C 180,E1 -28967.568,E2 -28967.568} C_VEL
LIN {X 0,Y 258.341,Z 962.868,A -85,B 0,C 180,E1 -28969.447,E2 -28969.447} C_VEL
LIN {X 0,Y 274.739,Z 944.791,A -85,B 0,C 180,E1 -28971.151,E2 -28971.151} C_VEL
LIN {X 0,Y 288.497,Z 927.813,A -85,B 0,C 180,E1 -28972.407,E2 -28972.407} C_VEL
LIN {X 0,Y 303.835,Z 906.367,A -85,B 0,C 180,E1 -28973.642,E2 -28973.642} C_VEL
LIN {X 0,Y 315.424,Z 887.837,A -85,B 0,C 180,E1 -28974.487,E2 -28974.487} C_VEL
LIN {X 0,Y 327.359,Z 866.103,A -85,B 0,C 180,E1 -28975.269,E2 -28975.269} C_VEL
LIN {X 0,Y 336.847,Z 845.738,A -85,B 0,C 180,E1 -28975.846,E2 -28975.846} C_VEL
LIN {X 0,Y 345.88,Z 823.129,A -85,B 0,C 180,E1 -28976.354,E2 -28976.354} C_VEL
LIN {X 0,Y 353.607,Z 798.995,A -85,B 0,C 180,E1 -28976.76,E2 -28976.76} C_VEL
LIN {X 0,Y 359.399,Z 776.228,A -85,B 0,C 180,E1 -28977.068,E2 -28977.068} C_VEL
LIN {X 0,Y 364.01,Z 750.794,A -85,B 0,C 180,E1 -28977.383,E2 -28977.383} C_VEL
LIN {X 0,Y 374.357,Z 666.292,A -85,B 0,C 180,E1 -28978.385,E2 -28978.385} C_VEL
LIN {X 0,Y 374.323,Z 665.024,A -85,B 0,C 180,E1 -28980.306,E2 -28980.306} C_VEL
LIN {X 0,Y 374.328,Z 666.477,A -85,B 0,C 180,E1 -28982.006,E2 -28982.006} C_VEL
LIN {X 0,Y 363.684,Z 752.807,A -85,B 0,C 180,E1 -28983.004,E2 -28983.004} C_VEL
LIN {X 0,Y 358.72,Z 778.521,A -85,B 0,C 180,E1 -28983.338,E2 -28983.338} C_VEL
LIN {X 0,Y 353.065,Z 800.251,A -85,B 0,C 180,E1 -28983.687,E2 -28983.687} C_VEL
LIN {X 0,Y 344.89,Z 824.951,A -85,B 0,C 180,E1 -28984.207,E2 -28984.207} C_VEL
LIN {X 0,Y 336.621,Z 845.427,A -85,B 0,C 180,E1 -28984.757,E2 -28984.757} C_VEL
LIN {X 0,Y 325.964,Z 867.867,A -85,B 0,C 180,E1 -28985.501,E2 -28985.501} C_VEL
LIN {X 0,Y 314.878,Z 887.684,A -85,B 0,C 180,E1 -28986.32,E2 -28986.32} C_VEL
LIN {X 0,Y 301.95,Z 908.068,A -85,B 0,C 180,E1 -28987.354,E2 -28987.354} C_VEL
LIN {X 0,Y 287.982,Z 927.086,A -85,B 0,C 180,E1 -28988.586,E2 -28988.586} C_VEL
LIN {X 0,Y 273.674,Z 944.515,A -85,B 0,C 180,E1 -28989.989,E2 -28989.989} C_VEL
LIN {X 0,Y 257.399,Z 962.017,A -85,B 0,C 180,E1 -28991.787,E2 -28991.787} C_VEL
LIN {X 0,Y 242.81,Z 976.085,A -85,B 0,C 180,E1 -28993.629,E2 -28993.629} C_VEL
LIN {X 0,Y 224.92,Z 991.632,A -85,B 0,C 180,E1 -28996.264,E2 -28996.264} C_VEL
LIN {X 0,Y 208.509,Z 1004.292,A -85,B 0,C 180,E1 -28999.145,E2 -28999.145} C_VEL
LIN {X 0,Y 191.027,Z 1016.602,A -85,B 0,C 180,E1 -29002.893,E2 -29002.893} C_VEL
LIN {X 0,Y 173.705,Z 1027.406,A -85,B 0,C 180,E1 -29007.568,E2 -29007.568} C_VEL
LIN {X 0,Y 157.722,Z 1036.602,A -85,B 0,C 180,E1 -29013.194,E2 -29013.194} C_VEL
LIN {X 0,Y 142.25,Z 1044.681,A -85,B 0,C 180,E1 -29020.612,E2 -29020.612} C_VEL
LIN {X 0,Y 130.399,Z 1050.592,A -85,B 0,C 180,E1 -29028.743,E2 -29028.743} C_VEL
LIN {X 0,Y 120.299,Z 1055.539,A -85,B 0,C 180,E1 -29039.535,E2 -29039.535} C_VEL
LIN {X 0,Y 114.96,Z 1058.34,A -85,B 0,C 180,E1 -29049.641,E2 -29049.641} C_VEL
LIN {X 0,Y 112.504,Z 1060.003,A -85,B 0,C 180,E1 -29060.279,E2 -29060.279} C_VEL
LIN {X 0,Y 112.064,Z 1060.497,A -85,B 0,C 180,E1 -29069.489,E2 -29069.489} C_VEL
LIN {X 0,Y 112.386,Z 1060.16,A -85,B 0,C 180,E1 -29078.7,E2 -29078.7} C_VEL
LIN {X 0,Y 114.755,Z 1058.501,A -85,B 0,C 180,E1 -29089.866,E2 -29089.866} C_VEL
LIN {X 0,Y 119.929,Z 1055.765,A -85,B 0,C 180,E1 -29100.016,E2 -29100.016} C_VEL
LIN {X 0,Y 129.86,Z 1050.951,A -85,B 0,C 180,E1 -29110.881,E2 -29110.881} C_VEL
LIN {X 0,Y 141.581,Z 1045.11,A -85,B 0,C 180,E1 -29119.084,E2 -29119.084} C_VEL
LIN {X 0,Y 156.265,Z 1037.543,A -85,B 0,C 180,E1 -29126.287,E2 -29126.287} C_VEL
LIN {X 0,Y 172.862,Z 1028.05,A -85,B 0,C 180,E1 -29132.252,E2 -29132.252} C_VEL
LIN {X 0,Y 190.131,Z 1017.345,A -85,B 0,C 180,E1 -29136.973,E2 -29136.973} C_VEL
LIN {X 0,Y 207.579,Z 1005.182,A -85,B 0,C 180,E1 -29140.755,E2 -29140.755} C_VEL
LIN {X 0,Y 223.135,Z 993.268,A -85,B 0,C 180,E1 -29143.528,E2 -29143.528} C_VEL
LIN {X 0,Y 241.839,Z 977.268,A -85,B 0,C 180,E1 -29146.317,E2 -29146.317} C_VEL
LIN {X 0,Y 256.415,Z 963.31,A -85,B 0,C 180,E1 -29148.175,E2 -29148.175} C_VEL
LIN {X 0,Y 273.098,Z 945.572,A -85,B 0,C 180,E1 -29150.026,E2 -29150.026} C_VEL
LIN {X 0,Y 287.659,Z 927.919,A -85,B 0,C 180,E1 -29151.46,E2 -29151.46} C_VEL
LIN {X 0,Y 301.903,Z 908.627,A -85,B 0,C 180,E1 -29152.717,E2 -29152.717} C_VEL
LIN {X 0,Y 314.837,Z 888.323,A -85,B 0,C 180,E1 -29153.751,E2 -29153.751} C_VEL
LIN {X 0,Y 325.927,Z 868.56,A -85,B 0,C 180,E1 -29154.571,E2 -29154.571} C_VEL
LIN {X 0,Y 336.589,Z 846.29,A -85,B 0,C 180,E1 -29155.313,E2 -29155.313} C_VEL
LIN {X 0,Y 344.861,Z 825.932,A -85,B 0,C 180,E1 -29155.864,E2 -29155.864} C_VEL
LIN {X 0,Y 353.315,Z 800.587,A -85,B 0,C 180,E1 -29156.401,E2 -29156.401} C_VEL
LIN {X 0,Y 359.006,Z 778.773,A -85,B 0,C 180,E1 -29156.752,E2 -29156.752} C_VEL
LIN {X 0,Y 363.948,Z 753.392,A -85,B 0,C 180,E1 -29157.082,E2 -29157.082} C_VEL
LIN {X 0,Y 373.22,Z 678.604,A -85,B 0,C 180,E1 -29157.947,E2 -29157.947} C_VEL
LIN {X 0,Y 374.663,Z 666.562,A -85,B 0,C 180,E1 -29158.123,E2 -29158.123} C_VEL
LIN {X 0,Y 374.623,Z 665.537,A -85,B 0,C 180,E1 -29160,E2 -29160} C_VEL
LIN {X 0,Y 374.642,Z 666.892,A -85,B 0,C 180,E1 -29161.643,E2 -29161.643} C_VEL
LIN {X 0,Y 363.928,Z 753.813,A -85,B 0,C 180,E1 -29162.65,E2 -29162.65} C_VEL
LIN {X 0,Y 358.928,Z 779.688,A -85,B 0,C 180,E1 -29162.974,E2 -29162.974} C_VEL
LIN {X 0,Y 353.164,Z 801.769,A -85,B 0,C 180,E1 -29163.276,E2 -29163.276} C_VEL
LIN {X 0,Y 344.689,Z 827.145,A -85,B 0,C 180,E1 -29163.721,E2 -29163.721} C_VEL
LIN {X 0,Y 336.364,Z 847.634,A -85,B 0,C 180,E1 -29164.194,E2 -29164.194} C_VEL
LIN {X 0,Y 325.145,Z 870.981,A -85,B 0,C 180,E1 -29164.883,E2 -29164.883} C_VEL
LIN {X 0,Y 314.464,Z 890.014,A -85,B 0,C 180,E1 -29165.595,E2 -29165.595} C_VEL
LIN {X 0,Y 301.364,Z 910.636,A -85,B 0,C 180,E1 -29166.563,E2 -29166.563} C_VEL
LIN {X 0,Y 287.075,Z 930.051,A -85,B 0,C 180,E1 -29167.726,E2 -29167.726} C_VEL
LIN {X 0,Y 282.464,Z 935.989,A -85,B 0,C 180,E1 -29168.139,E2 -29168.139} C_VEL
LIN {X 0,Y 277.563,Z 941.904,A -85,B 0,C 180,E1 -29168.379,E2 -29168.379} C_VEL
LIN {X 0,Y 263.612,Z 956.415,A -85,B 0,C 180,E1 -29168.342,E2 -29168.342} C_VEL
LIN {X 0,Y 258.17,Z 961.767,A -85,B 0,C 180,E1 -29168.645,E2 -29168.645} C_VEL
LIN {X 0,Y 241.966,Z 977.394,A -85,B 0,C 180,E1 -29170.422,E2 -29170.422} C_VEL
LIN {X 0,Y 224.458,Z 992.678,A -85,B 0,C 180,E1 -29172.689,E2 -29172.689} C_VEL
LIN {X 0,Y 206.477,Z 1006.544,A -85,B 0,C 180,E1 -29175.488,E2 -29175.488} C_VEL
LIN {X 0,Y 189.941,Z 1018.113,A -85,B 0,C 180,E1 -29178.637,E2 -29178.637} C_VEL
LIN {X 0,Y 170.042,Z 1030.602,A -85,B 0,C 180,E1 -29183.462,E2 -29183.462} C_VEL
LIN {X 0,Y 154.573,Z 1039.395,A -85,B 0,C 180,E1 -29188.388,E2 -29188.388} C_VEL
LIN {X 0,Y 137.157,Z 1048.504,A -85,B 0,C 180,E1 -29195.981,E2 -29195.981} C_VEL
LIN {X 0,Y 124.18,Z 1054.848,A -85,B 0,C 180,E1 -29204.223,E2 -29204.223} C_VEL
LIN {X 0,Y 112.935,Z 1060.369,A -85,B 0,C 180,E1 -29215.484,E2 -29215.484} C_VEL
LIN {X 0,Y 106.753,Z 1063.651,A -85,B 0,C 180,E1 -29226.834,E2 -29226.834} C_VEL
LIN {X 0,Y 104.276,Z 1065.504,A -85,B 0,C 180,E1 -29237.821,E2 -29237.821} C_VEL
LIN {X 0,Y 104.02,Z 1066.154,A -85,B 0,C 180,E1 -29246.693,E2 -29246.693} C_VEL
LIN {X 0,Y 104.027,Z 1066.172,A -85,B 0,C 180,E1 -29252.754,E2 -29252.754} C_VEL
LIN {X 0,Y 104.225,Z 1065.557,A -85,B 0,C 180,E1 -29261.622,E2 -29261.622} C_VEL
LIN {X 0,Y 106.558,Z 1063.738,A -85,B 0,C 180,E1 -29272.626,E2 -29272.626} C_VEL
LIN {X 0,Y 112.571,Z 1060.489,A -85,B 0,C 180,E1 -29284.027,E2 -29284.027} C_VEL
LIN {X 0,Y 123.645,Z 1055.036,A -85,B 0,C 180,E1 -29295.368,E2 -29295.368} C_VEL
LIN {X 0,Y 136.193,Z 1048.877,A -85,B 0,C 180,E1 -29303.51,E2 -29303.51} C_VEL
LIN {X 0,Y 153.824,Z 1039.686,A -85,B 0,C 180,E1 -29311.345,E2 -29311.345} C_VEL
LIN {X 0,Y 170.032,Z 1030.467,A -85,B 0,C 180,E1 -29316.544,E2 -29316.544} C_VEL
LIN {X 0,Y 189.931,Z 1017.942,A -85,B 0,C 180,E1 -29321.37,E2 -29321.37} C_VEL
LIN {X 0,Y 206.467,Z 1006.349,A -85,B 0,C 180,E1 -29324.52,E2 -29324.52} C_VEL
LIN {X 0,Y 225.359,Z 991.654,A -85,B 0,C 180,E1 -29327.45,E2 -29327.45} C_VEL
LIN {X 0,Y 241.957,Z 977.122,A -85,B 0,C 180,E1 -29329.588,E2 -29329.588} C_VEL
LIN {X 0,Y 259.355,Z 960.236,A -85,B 0,C 180,E1 -29331.486,E2 -29331.486} C_VEL
LIN {X 0,Y 275.036,Z 942.893,A -85,B 0,C 180,E1 -29332.97,E2 -29332.97} C_VEL
LIN {X 0,Y 289.467,Z 925.143,A -85,B 0,C 180,E1 -29334.166,E2 -29334.166} C_VEL
LIN {X 0,Y 304.016,Z 904.669,A -85,B 0,C 180,E1 -29335.236,E2 -29335.236} C_VEL
LIN {X 0,Y 316.216,Z 885.171,A -85,B 0,C 180,E1 -29336.049,E2 -29336.049} C_VEL
LIN {X 0,Y 328.48,Z 862.413,A -85,B 0,C 180,E1 -29336.784,E2 -29336.784} C_VEL
LIN {X 0,Y 337.674,Z 842.493,A -85,B 0,C 180,E1 -29337.284,E2 -29337.284} C_VEL
LIN {X 0,Y 347.224,Z 817.83,A -85,B 0,C 180,E1 -29337.77,E2 -29337.77} C_VEL
LIN {X 0,Y 353.968,Z 796.227,A -85,B 0,C 180,E1 -29338.095,E2 -29338.095} C_VEL
LIN {X 0,Y 360.099,Z 771.254,A -85,B 0,C 180,E1 -29338.405,E2 -29338.405} C_VEL
LIN {X 0,Y 364.118,Z 747.875,A -85,B 0,C 180,E1 -29338.678,E2 -29338.678} C_VEL
LIN {X 0,Y 373.312,Z 673.46,A -85,B 0,C 180,E1 -29339.54,E2 -29339.54} C_VEL
LIN {X 0,Y 373.342,Z 673.015,A -85,B 0,C 180,E1 -29340.307,E2 -29340.307} C_VEL
LIN {X 0,Y 373.296,Z 673.577,A -85,B 0,C 180,E1 -29340.857,E2 -29340.857} C_VEL
LIN {X 0,Y 363.325,Z 753.235,A -85,B 0,C 180,E1 -29341.746,E2 -29341.746} C_VEL
LIN {X 0,Y 358.34,Z 778.759,A -85,B 0,C 180,E1 -29342.059,E2 -29342.059} C_VEL
LIN {X 0,Y 352.624,Z 800.533,A -85,B 0,C 180,E1 -29342.389,E2 -29342.389} C_VEL
LIN {X 0,Y 344.395,Z 825.174,A -85,B 0,C 180,E1 -29342.876,E2 -29342.876} C_VEL
LIN {X 0,Y 336.05,Z 845.648,A -85,B 0,C 180,E1 -29343.392,E2 -29343.392} C_VEL
LIN {X 0,Y 325.291,Z 868.088,A -85,B 0,C 180,E1 -29344.089,E2 -29344.089} C_VEL
LIN {X 0,Y 314.092,Z 887.905,A -85,B 0,C 180,E1 -29344.857,E2 -29344.857} C_VEL
LIN {X 0,Y 301.154,Z 908.09,A -85,B 0,C 180,E1 -29345.818,E2 -29345.818} C_VEL
LIN {X 0,Y 286.537,Z 927.744,A -85,B 0,C 180,E1 -29347.015,E2 -29347.015} C_VEL
LIN {X 0,Y 271.857,Z 945.348,A -85,B 0,C 180,E1 -29348.358,E2 -29348.358} C_VEL
LIN {X 0,Y 254.925,Z 963.155,A -85,B 0,C 180,E1 -29350.104,E2 -29350.104} C_VEL
LIN {X 0,Y 239.179,Z 977.98,A -85,B 0,C 180,E1 -29351.976,E2 -29351.976} C_VEL
LIN {X 0,Y 220.124,Z 993.892,A -85,B 0,C 180,E1 -29354.641,E2 -29354.641} C_VEL
LIN {X 0,Y 204.222,Z 1005.768,A -85,B 0,C 180,E1 -29357.306,E2 -29357.306} C_VEL
LIN {X 0,Y 184.646,Z 1018.876,A -85,B 0,C 180,E1 -29361.345,E2 -29361.345} C_VEL
LIN {X 0,Y 168.483,Z 1028.529,A -85,B 0,C 180,E1 -29365.57,E2 -29365.57} C_VEL
LIN {X 0,Y 151.035,Z 1038.043,A -85,B 0,C 180,E1 -29371.534,E2 -29371.534} C_VEL
LIN {X 0,Y 135.791,Z 1045.493,A -85,B 0,C 180,E1 -29378.692,E2 -29378.692} C_VEL
LIN {X 0,Y 122.331,Z 1051.784,A -85,B 0,C 180,E1 -29387.915,E2 -29387.915} C_VEL
LIN {X 0,Y 112.293,Z 1056.219,A -85,B 0,C 180,E1 -29398.906,E2 -29398.906} C_VEL
LIN {X 0,Y 106.618,Z 1058.993,A -85,B 0,C 180,E1 -29410.269,E2 -29410.269} C_VEL
LIN {X 0,Y 104.303,Z 1060.434,A -85,B 0,C 180,E1 -29422.288,E2 -29422.288} C_VEL
LIN {X 0,Y 104.068,Z 1060.698,A -85,B 0,C 180,E1 -29431.102,E2 -29431.102} C_VEL
LIN {X 0,Y 104.63,Z 1060.184,A -85,B 0,C 180,E1 -29441.019,E2 -29441.019} C_VEL
LIN {X 0,Y 107.363,Z 1058.608,A -85,B 0,C 180,E1 -29451.872,E2 -29451.872} C_VEL
LIN {X 0,Y 113.288,Z 1055.828,A -85,B 0,C 180,E1 -29462.575,E2 -29462.575} C_VEL
LIN {X 0,Y 124.807,Z 1050.673,A -85,B 0,C 180,E1 -29474.187,E2 -29474.187} C_VEL
LIN {X 0,Y 136.968,Z 1045.032,A -85,B 0,C 180,E1 -29482.038,E2 -29482.038} C_VEL
LIN {X 0,Y 153.297,Z 1036.997,A -85,B 0,C 180,E1 -29489.427,E2 -29489.427} C_VEL
LIN {X 0,Y 169.977,Z 1027.816,A -85,B 0,C 180,E1 -29494.946,E2 -29494.946} C_VEL
LIN {X 0,Y 187.91,Z 1017.048,A -85,B 0,C 180,E1 -29499.475,E2 -29499.475} C_VEL
LIN {X 0,Y 205.897,Z 1004.771,A -85,B 0,C 180,E1 -29503.075,E2 -29503.075} C_VEL
LIN {X 0,Y 223.654,Z 991.405,A -85,B 0,C 180,E1 -29505.965,E2 -29505.965} C_VEL
LIN {X 0,Y 240.959,Z 976.646,A -85,B 0,C 180,E1 -29508.326,E2 -29508.326} C_VEL
LIN {X 0,Y 256.201,Z 962.218,A -85,B 0,C 180,E1 -29510.112,E2 -29510.112} C_VEL
LIN {X 0,Y 274.067,Z 943.16,A -85,B 0,C 180,E1 -29511.93,E2 -29511.93} C_VEL
LIN {X 0,Y 288.004,Z 926.319,A -85,B 0,C 180,E1 -29513.185,E2 -29513.185} C_VEL
LIN {X 0,Y 303.399,Z 905.214,A -85,B 0,C 180,E1 -29514.432,E2 -29514.432} C_VEL
LIN {X 0,Y 315.033,Z 886.918,A -85,B 0,C 180,E1 -29515.284,E2 -29515.284} C_VEL
LIN {X 0,Y 327.217,Z 865.059,A -85,B 0,C 180,E1 -29516.114,E2 -29516.114} C_VEL
LIN {X 0,Y 337.009,Z 844.245,A -85,B 0,C 180,E1 -29516.741,E2 -29516.741} C_VEL
LIN {X 0,Y 345.36,Z 823.577,A -85,B 0,C 180,E1 -29517.252,E2 -29517.252} C_VEL
LIN {X 0,Y 353.407,Z 799.019,A -85,B 0,C 180,E1 -29517.73,E2 -29517.73} C_VEL
LIN {X 0,Y 359.105,Z 777.023,A -85,B 0,C 180,E1 -29518.058,E2 -29518.058} C_VEL
LIN {X 0,Y 364.029,Z 750.805,A -85,B 0,C 180,E1 -29518.373,E2 -29518.373} C_VEL
LIN {X 0,Y 373.623,Z 673.835,A -85,B 0,C 180,E1 -29519.233,E2 -29519.233} C_VEL
LIN {X 0,Y 373.643,Z 673.519,A -85,B 0,C 180,E1 -29520,E2 -29520} C_VEL
LIN {X 0,Y 373.595,Z 674.099,A -85,B 0,C 180,E1 -29520.497,E2 -29520.497} C_VEL
LIN {X 0,Y 363.599,Z 753.941,A -85,B 0,C 180,E1 -29521.39,E2 -29521.39} C_VEL
LIN {X 0,Y 358.557,Z 779.673,A -85,B 0,C 180,E1 -29521.695,E2 -29521.695} C_VEL
LIN {X 0,Y 352.734,Z 801.782,A -85,B 0,C 180,E1 -29521.976,E2 -29521.976} C_VEL
LIN {X 0,Y 344.261,Z 826.938,A -85,B 0,C 180,E1 -29522.384,E2 -29522.384} C_VEL
LIN {X 0,Y 335.871,Z 847.426,A -85,B 0,C 180,E1 -29522.822,E2 -29522.822} C_VEL
LIN {X 0,Y 324.557,Z 870.771,A -85,B 0,C 180,E1 -29523.461,E2 -29523.461} C_VEL
LIN {X 0,Y 313.777,Z 889.803,A -85,B 0,C 180,E1 -29524.12,E2 -29524.12} C_VEL
LIN {X 0,Y 300.62,Z 910.316,A -85,B 0,C 180,E1 -29525.018,E2 -29525.018} C_VEL
LIN {X 0,Y 286.208,Z 929.692,A -85,B 0,C 180,E1 -29526.099,E2 -29526.099} C_VEL
LIN {X 0,Y 271.22,Z 947.73,A -85,B 0,C 180,E1 -29527.384,E2 -29527.384} C_VEL
LIN {X 0,Y 258.17,Z 961.767,A -85,B 0,C 180,E1 -29528.645,E2 -29528.645} C_VEL
LIN {X 0,Y 252.643,Z 967.053,A -85,B 0,C 180,E1 -29528.974,E2 -29528.974} C_VEL
LIN {X 0,Y 237.469,Z 980.261,A -85,B 0,C 180,E1 -29529.108,E2 -29529.108} C_VEL
LIN {X 0,Y 231.647,Z 985.08,A -85,B 0,C 180,E1 -29529.515,E2 -29529.515} C_VEL
LIN {X 0,Y 214.468,Z 998.894,A -85,B 0,C 180,E1 -29531.745,E2 -29531.745} C_VEL
LIN {X 0,Y 195.429,Z 1012.665,A -85,B 0,C 180,E1 -29534.76,E2 -29534.76} C_VEL
LIN {X 0,Y 177.042,Z 1024.4,A -85,B 0,C 180,E1 -29538.409,E2 -29538.409} C_VEL
LIN {X 0,Y 158.729,Z 1035.041,A -85,B 0,C 180,E1 -29543.117,E2 -29543.117} C_VEL
LIN {X 0,Y 140.747,Z 1044.26,A -85,B 0,C 180,E1 -29549.353,E2 -29549.353} C_VEL
LIN {X 0,Y 124.57,Z 1052.004,A -85,B 0,C 180,E1 -29557.377,E2 -29557.377} C_VEL
LIN {X 0,Y 111.143,Z 1057.917,A -85,B 0,C 180,E1 -29567.566,E2 -29567.566} C_VEL
LIN {X 0,Y 101.963,Z 1062.143,A -85,B 0,C 180,E1 -29579.34,E2 -29579.34} C_VEL
LIN {X 0,Y 96.914,Z 1064.852,A -85,B 0,C 180,E1 -29593.208,E2 -29593.208} C_VEL
LIN {X 0,Y 96.01,Z 1065.815,A -85,B 0,C 180,E1 -29603.421,E2 -29603.421} C_VEL
LIN {X 0,Y 96.05,Z 1066.03,A -85,B 0,C 180,E1 -29611.192,E2 -29611.192} C_VEL
LIN {X 0,Y 96.153,Z 1065.557,A -85,B 0,C 180,E1 -29620.788,E2 -29620.788} C_VEL
LIN {X 0,Y 98.638,Z 1063.758,A -85,B 0,C 180,E1 -29633.287,E2 -29633.287} C_VEL
LIN {X 0,Y 104.691,Z 1060.768,A -85,B 0,C 180,E1 -29644.963,E2 -29644.963} C_VEL
LIN {X 0,Y 116.304,Z 1055.599,A -85,B 0,C 180,E1 -29656.95,E2 -29656.95} C_VEL
LIN {X 0,Y 129.743,Z 1049.433,A -85,B 0,C 180,E1 -29665.549,E2 -29665.549} C_VEL
LIN {X 0,Y 146.193,Z 1041.512,A -85,B 0,C 180,E1 -29672.764,E2 -29672.764} C_VEL
LIN {X 0,Y 164.422,Z 1031.643,A -85,B 0,C 180,E1 -29678.501,E2 -29678.501} C_VEL
LIN {X 0,Y 183.082,Z 1020.588,A -85,B 0,C 180,E1 -29682.891,E2 -29682.891} C_VEL
LIN {X 0,Y 201.703,Z 1008.055,A -85,B 0,C 180,E1 -29686.316,E2 -29686.316} C_VEL
LIN {X 0,Y 219.075,Z 995.129,A -85,B 0,C 180,E1 -29688.899,E2 -29688.899} C_VEL
LIN {X 0,Y 237.772,Z 979.459,A -85,B 0,C 180,E1 -29691.2,E2 -29691.2} C_VEL
LIN {X 0,Y 252.974,Z 965.225,A -85,B 0,C 180,E1 -29692.786,E2 -29692.786} C_VEL
LIN {X 0,Y 270.284,Z 947.143,A -85,B 0,C 180,E1 -29694.346,E2 -29694.346} C_VEL
LIN {X 0,Y 285.335,Z 929.207,A -85,B 0,C 180,E1 -29695.531,E2 -29695.531} C_VEL
LIN {X 0,Y 300.362,Z 909.09,A -85,B 0,C 180,E1 -29696.565,E2 -29696.565} C_VEL
LIN {X 0,Y 313.294,Z 889.024,A -85,B 0,C 180,E1 -29697.372,E2 -29697.372} C_VEL
LIN {X 0,Y 325.155,Z 868.129,A -85,B 0,C 180,E1 -29698.031,E2 -29698.031} C_VEL
LIN {X 0,Y 335.723,Z 846.072,A -85,B 0,C 180,E1 -29698.573,E2 -29698.573} C_VEL
LIN {X 0,Y 344.564,Z 824.407,A -85,B 0,C 180,E1 -29698.992,E2 -29698.992} C_VEL
LIN {X 0,Y 352.79,Z 799.497,A -85,B 0,C 180,E1 -29699.353,E2 -29699.353} C_VEL
LIN {X 0,Y 358.53,Z 777.47,A -85,B 0,C 180,E1 -29699.611,E2 -29699.611} C_VEL
LIN {X 0,Y 363.522,Z 751.073,A -85,B 0,C 180,E1 -29699.905,E2 -29699.905} C_VEL
LIN {X 0,Y 366.856,Z 725.835,A -85,B 0,C 180,E1 -29700.185,E2 -29700.185} C_VEL
LIN {X 0,Y 362.132,Z 759.662,A -85,B 0,C 180,E1 -29700.552,E2 -29700.552} C_VEL
LIN {X 0,Y 357.409,Z 782.052,A -85,B 0,C 180,E1 -29700.82,E2 -29700.82} C_VEL
LIN {X 0,Y 350.784,Z 806.158,A -85,B 0,C 180,E1 -29701.177,E2 -29701.177} C_VEL
LIN {X 0,Y 343.094,Z 827.957,A -85,B 0,C 180,E1 -29701.595,E2 -29701.595} C_VEL
LIN {X 0,Y 334.189,Z 849.247,A -85,B 0,C 180,E1 -29702.11,E2 -29702.11} C_VEL
LIN {X 0,Y 322.847,Z 871.892,A -85,B 0,C 180,E1 -29702.793,E2 -29702.793} C_VEL
LIN {X 0,Y 311.968,Z 890.669,A -85,B 0,C 180,E1 -29703.491,E2 -29703.491} C_VEL
LIN {X 0,Y 297.384,Z 912.517,A -85,B 0,C 180,E1 -29704.502,E2 -29704.502} C_VEL
LIN {X 0,Y 284.282,Z 929.686,A -85,B 0,C 180,E1 -29705.512,E2 -29705.512} C_VEL
LIN {X 0,Y 268.799,Z 947.797,A -85,B 0,C 180,E1 -29706.836,E2 -29706.836} C_VEL
LIN {X 0,Y 252.25,Z 964.706,A -85,B 0,C 180,E1 -29708.434,E2 -29708.434} C_VEL
LIN {X 0,Y 234.821,Z 980.706,A -85,B 0,C 180,E1 -29710.387,E2 -29710.387} C_VEL
LIN {X 0,Y 216.372,Z 995.498,A -85,B 0,C 180,E1 -29712.824,E2 -29712.824} C_VEL
LIN {X 0,Y 198.38,Z 1008.498,A -85,B 0,C 180,E1 -29715.701,E2 -29715.701} C_VEL
LIN {X 0,Y 179.258,Z 1020.619,A -85,B 0,C 180,E1 -29719.496,E2 -29719.496} C_VEL
LIN {X 0,Y 161.869,Z 1030.555,A -85,B 0,C 180,E1 -29723.906,E2 -29723.906} C_VEL
LIN {X 0,Y 143.382,Z 1039.906,A -85,B 0,C 180,E1 -29730.149,E2 -29730.149} C_VEL
LIN {X 0,Y 128.205,Z 1046.899,A -85,B 0,C 180,E1 -29737.297,E2 -29737.297} C_VEL
LIN {X 0,Y 113.771,Z 1053.005,A -85,B 0,C 180,E1 -29747.412,E2 -29747.412} C_VEL
LIN {X 0,Y 104.656,Z 1056.746,A -85,B 0,C 180,E1 -29757.655,E2 -29757.655} C_VEL
LIN {X 0,Y 98.206,Z 1059.625,A -85,B 0,C 180,E1 -29771.244,E2 -29771.244} C_VEL
LIN {X 0,Y 96.259,Z 1060.689,A -85,B 0,C 180,E1 -29782.84,E2 -29782.84} C_VEL
LIN {X 0,Y 96.074,Z 1060.889,A -85,B 0,C 180,E1 -29791.79,E2 -29791.79} C_VEL
LIN {X 0,Y 96.825,Z 1060.334,A -85,B 0,C 180,E1 -29802.525,E2 -29802.525} C_VEL
LIN {X 0,Y 100.111,Z 1058.716,A -85,B 0,C 180,E1 -29814.174,E2 -29814.174} C_VEL
LIN {X 0,Y 107.298,Z 1055.738,A -85,B 0,C 180,E1 -29825.951,E2 -29825.951} C_VEL
LIN {X 0,Y 119.757,Z 1050.588,A -85,B 0,C 180,E1 -29837.445,E2 -29837.445} C_VEL
LIN {X 0,Y 133.419,Z 1044.659,A -85,B 0,C 180,E1 -29845.526,E2 -29845.526} C_VEL
LIN {X 0,Y 151.57,Z 1036.021,A -85,B 0,C 180,E1 -29852.947,E2 -29852.947} C_VEL
LIN {X 0,Y 167.481,Z 1027.583,A -85,B 0,C 180,E1 -29857.726,E2 -29857.726} C_VEL
LIN {X 0,Y 186.919,Z 1016.141,A -85,B 0,C 180,E1 -29862.211,E2 -29862.211} C_VEL
LIN {X 0,Y 204.557,Z 1004.36,A -85,B 0,C 180,E1 -29865.43,E2 -29865.43} C_VEL
LIN {X 0,Y 222.731,Z 990.925,A -85,B 0,C 180,E1 -29868.141,E2 -29868.141} C_VEL
LIN {X 0,Y 240.376,Z 976.023,A -85,B 0,C 180,E1 -29870.349,E2 -29870.349} C_VEL
LIN {X 0,Y 256.428,Z 960.984,A -85,B 0,C 180,E1 -29872.065,E2 -29872.065} C_VEL
LIN {X 0,Y 273.639,Z 942.693,A -85,B 0,C 180,E1 -29873.67,E2 -29873.67} C_VEL
LIN {X 0,Y 287.4,Z 926.226,A -85,B 0,C 180,E1 -29874.81,E2 -29874.81} C_VEL
LIN {X 0,Y 303.21,Z 904.694,A -85,B 0,C 180,E1 -29875.988,E2 -29875.988} C_VEL
LIN {X 0,Y 314.963,Z 886.32,A -85,B 0,C 180,E1 -29876.781,E2 -29876.781} C_VEL
LIN {X 0,Y 327.263,Z 864.267,A -85,B 0,C 180,E1 -29877.554,E2 -29877.554} C_VEL
LIN {X 0,Y 337.142,Z 843.326,A -85,B 0,C 180,E1 -29878.135,E2 -29878.135} C_VEL
LIN {X 0,Y 346.334,Z 820.45,A -85,B 0,C 180,E1 -29878.648,E2 -29878.648} C_VEL
LIN {X 0,Y 353.803,Z 797.055,A -85,B 0,C 180,E1 -29879.062,E2 -29879.062} C_VEL
LIN {X 0,Y 359.981,Z 772.727,A -85,B 0,C 180,E1 -29879.392,E2 -29879.392} C_VEL
LIN {X 0,Y 364.283,Z 748.298,A -85,B 0,C 180,E1 -29879.662,E2 -29879.662} C_VEL
LIN {X 0,Y 366.697,Z 730.081,A -85,B 0,C 180,E1 -29879.867,E2 -29879.867} C_VEL
LIN {X 0,Y 361.995,Z 762.307,A -85,B 0,C 180,E1 -29880.219,E2 -29880.219} C_VEL
LIN {X 0,Y 357.223,Z 784.438,A -85,B 0,C 180,E1 -29880.468,E2 -29880.468} C_VEL
LIN {X 0,Y 349.721,Z 810.573,A -85,B 0,C 180,E1 -29880.797,E2 -29880.797} C_VEL
LIN {X 0,Y 342.527,Z 830.594,A -85,B 0,C 180,E1 -29881.112,E2 -29881.112} C_VEL
LIN {X 0,Y 332.592,Z 853.815,A -85,B 0,C 180,E1 -29881.592,E2 -29881.592} C_VEL
LIN {X 0,Y 322.19,Z 874.176,A -85,B 0,C 180,E1 -29882.139,E2 -29882.139} C_VEL
LIN {X 0,Y 310.343,Z 894.483,A -85,B 0,C 180,E1 -29882.823,E2 -29882.823} C_VEL
LIN {X 0,Y 296.585,Z 914.803,A -85,B 0,C 180,E1 -29883.696,E2 -29883.696} C_VEL
LIN {X 0,Y 282.872,Z 932.725,A -85,B 0,C 180,E1 -29884.663,E2 -29884.663} C_VEL
LIN {X 0,Y 265.462,Z 952.719,A -85,B 0,C 180,E1 -29886.074,E2 -29886.074} C_VEL
LIN {X 0,Y 250.115,Z 968.331,A -85,B 0,C 180,E1 -29887.504,E2 -29887.504} C_VEL
LIN {X 0,Y 231.647,Z 985.08,A -85,B 0,C 180,E1 -29889.515,E2 -29889.515} C_VEL
LIN {X 0,Y 225.719,Z 989.843,A -85,B 0,C 180,E1 -29889.959,E2 -29889.959} C_VEL
LIN {X 0,Y 208.498,Z 1002.166,A -85,B 0,C 180,E1 -29890.39,E2 -29890.39} C_VEL
LIN {X 0,Y 203.239,Z 1005.726,A -85,B 0,C 180,E1 -29890.901,E2 -29890.901} C_VEL
LIN {X 0,Y 185.315,Z 1017.674,A -85,B 0,C 180,E1 -29893.78,E2 -29893.78} C_VEL
LIN {X 0,Y 164.146,Z 1030.162,A -85,B 0,C 180,E1 -29898.144,E2 -29898.144} C_VEL
LIN {X 0,Y 147.119,Z 1039.101,A -85,B 0,C 180,E1 -29902.793,E2 -29902.793} C_VEL
LIN {X 0,Y 127.395,Z 1048.373,A -85,B 0,C 180,E1 -29910.303,E2 -29910.303} C_VEL
LIN {X 0,Y 113.255,Z 1054.407,A -85,B 0,C 180,E1 -29918.209,E2 -29918.209} C_VEL
LIN {X 0,Y 99.793,Z 1059.93,A -85,B 0,C 180,E1 -29930.114,E2 -29930.114} C_VEL
LIN {X 0,Y 91.925,Z 1063.215,A -85,B 0,C 180,E1 -29942.816,E2 -29942.816} C_VEL
LIN {X 0,Y 88.493,Z 1065.072,A -85,B 0,C 180,E1 -29955.606,E2 -29955.606} C_VEL
LIN {X 0,Y 88.023,Z 1065.751,A -85,B 0,C 180,E1 -29966.743,E2 -29966.743} C_VEL
LIN {X 0,Y 88.023,Z 1065.744,A -85,B 0,C 180,E1 -29973.255,E2 -29973.255} C_VEL
LIN {X 0,Y 88.494,Z 1065.052,A -85,B 0,C 180,E1 -29984.393,E2 -29984.393} C_VEL
LIN {X 0,Y 91.923,Z 1063.181,A -85,B 0,C 180,E1 -29997.184,E2 -29997.184} C_VEL
LIN {X 0,Y 100.706,Z 1059.546,A -85,B 0,C 180,E1 -30010.942,E2 -30010.942} C_VEL
LIN {X 0,Y 113.871,Z 1054.07,A -85,B 0,C 180,E1 -30022.211,E2 -30022.211} C_VEL
LIN {X 0,Y 129.575,Z 1047.348,A -85,B 0,C 180,E1 -30030.69,E2 -30030.69} C_VEL
LIN {X 0,Y 147.399,Z 1038.828,A -85,B 0,C 180,E1 -30037.303,E2 -30037.303} C_VEL
LIN {X 0,Y 165,Z 1029.555,A -85,B 0,C 180,E1 -30042.065,E2 -30042.065} C_VEL
LIN {X 0,Y 185.666,Z 1017.264,A -85,B 0,C 180,E1 -30046.293,E2 -30046.293} C_VEL
LIN {X 0,Y 202.682,Z 1005.903,A -85,B 0,C 180,E1 -30049.028,E2 -30049.028} C_VEL
LIN {X 0,Y 222.359,Z 991.209,A -85,B 0,C 180,E1 -30051.601,E2 -30051.601} C_VEL
LIN {X 0,Y 239.531,Z 976.678,A -85,B 0,C 180,E1 -30053.46,E2 -30053.46} C_VEL
LIN {X 0,Y 257.443,Z 959.787,A -85,B 0,C 180,E1 -30055.098,E2 -30055.098} C_VEL
LIN {X 0,Y 274.007,Z 941.891,A -85,B 0,C 180,E1 -30056.407,E2 -30056.407} C_VEL
LIN {X 0,Y 289.254,Z 923.477,A -85,B 0,C 180,E1 -30057.45,E2 -30057.45} C_VEL
LIN {X 0,Y 303.546,Z 903.562,A -85,B 0,C 180,E1 -30058.323,E2 -30058.323} C_VEL
LIN {X 0,Y 316.011,Z 883.914,A -85,B 0,C 180,E1 -30059.011,E2 -30059.011} C_VEL
LIN {X 0,Y 327.971,Z 861.969,A -85,B 0,C 180,E1 -30059.605,E2 -30059.605} C_VEL
LIN {X 0,Y 336.962,Z 842.803,A -85,B 0,C 180,E1 -30060.007,E2 -30060.007} C_VEL
LIN {X 0,Y 342.748,Z 828.735,A -85,B 0,C 180,E1 -30060.266,E2 -30060.266} C_VEL
LIN {X 0,Y 333.492,Z 850.595,A -85,B 0,C 180,E1 -30060.76,E2 -30060.76} C_VEL
LIN {X 0,Y 322.555,Z 872.112,A -85,B 0,C 180,E1 -30061.364,E2 -30061.364} C_VEL
LIN {X 0,Y 311.353,Z 891.261,A -85,B 0,C 180,E1 -30062.024,E2 -30062.024} C_VEL
LIN {X 0,Y 296.367,Z 913.401,A -85,B 0,C 180,E1 -30062.978,E2 -30062.978} C_VEL
LIN {X 0,Y 282.641,Z 931.115,A -85,B 0,C 180,E1 -30063.955,E2 -30063.955} C_VEL
LIN {X 0,Y 265.122,Z 950.953,A -85,B 0,C 180,E1 -30065.344,E2 -30065.344} C_VEL
LIN {X 0,Y 249.696,Z 966.35,A -85,B 0,C 180,E1 -30066.738,E2 -30066.738} C_VEL
LIN {X 0,Y 230.647,Z 983.225,A -85,B 0,C 180,E1 -30068.731,E2 -30068.731} C_VEL
LIN {X 0,Y 213.775,Z 996.412,A -85,B 0,C 180,E1 -30070.818,E2 -30070.818} C_VEL
LIN {X 0,Y 194.507,Z 1009.91,A -85,B 0,C 180,E1 -30073.694,E2 -30073.694} C_VEL
LIN {X 0,Y 175.481,Z 1021.539,A -85,B 0,C 180,E1 -30077.235,E2 -30077.235} C_VEL
LIN {X 0,Y 156.225,Z 1032.095,A -85,B 0,C 180,E1 -30081.869,E2 -30081.869} C_VEL
LIN {X 0,Y 137.903,Z 1040.819,A -85,B 0,C 180,E1 -30087.801,E2 -30087.801} C_VEL
LIN {X 0,Y 120.701,Z 1048.278,A -85,B 0,C 180,E1 -30095.725,E2 -30095.725} C_VEL
LIN {X 0,Y 106.26,Z 1053.825,A -85,B 0,C 180,E1 -30105.868,E2 -30105.868} C_VEL
LIN {X 0,Y 95.608,Z 1057.888,A -85,B 0,C 180,E1 -30118.473,E2 -30118.473} C_VEL
LIN {X 0,Y 89.77,Z 1060.134,A -85,B 0,C 180,E1 -30132.499,E2 -30132.499} C_VEL
LIN {X 0,Y 88.217,Z 1060.944,A -85,B 0,C 180,E1 -30143.492,E2 -30143.492} C_VEL
LIN {X 0,Y 88.084,Z 1061.08,A -85,B 0,C 180,E1 -30152.636,E2 -30152.636} C_VEL
LIN {X 0,Y 89.082,Z 1060.484,A -85,B 0,C 180,E1 -30164.297,E2 -30164.297} C_VEL
LIN {X 0,Y 93.069,Z 1058.81,A -85,B 0,C 180,E1 -30176.91,E2 -30176.91} C_VEL
LIN {X 0,Y 102.244,Z 1055.475,A -85,B 0,C 180,E1 -30190.288,E2 -30190.288} C_VEL
LIN {X 0,Y 115.468,Z 1050.367,A -85,B 0,C 180,E1 -30201.202,E2 -30201.202} C_VEL
LIN {X 0,Y 130.391,Z 1044.285,A -85,B 0,C 180,E1 -30209.189,E2 -30209.189} C_VEL
LIN {X 0,Y 148.812,Z 1035.842,A -85,B 0,C 180,E1 -30216.037,E2 -30216.037} C_VEL
LIN {X 0,Y 165.392,Z 1027.349,A -85,B 0,C 180,E1 -30220.581,E2 -30220.581} C_VEL
LIN {X 0,Y 186.357,Z 1015.227,A -85,B 0,C 180,E1 -30224.969,E2 -30224.969} C_VEL
LIN {X 0,Y 203.567,Z 1003.95,A -85,B 0,C 180,E1 -30227.813,E2 -30227.813} C_VEL
LIN {X 0,Y 223.096,Z 989.607,A -85,B 0,C 180,E1 -30230.455,E2 -30230.455} C_VEL
LIN {X 0,Y 240.095,Z 975.401,A -85,B 0,C 180,E1 -30232.379,E2 -30232.379} C_VEL
LIN {X 0,Y 257.842,Z 958.882,A -85,B 0,C 180,E1 -30234.093,E2 -30234.093} C_VEL
LIN {X 0,Y 274.323,Z 941.253,A -85,B 0,C 180,E1 -30235.482,E2 -30235.482} C_VEL
LIN {X 0,Y 289.841,Z 922.666,A -85,B 0,C 180,E1 -30236.638,E2 -30236.638} C_VEL
LIN {X 0,Y 303.739,Z 903.443,A -85,B 0,C 180,E1 -30237.576,E2 -30237.576} C_VEL
LIN {X 0,Y 315.604,Z 884.915,A -85,B 0,C 180,E1 -30238.305,E2 -30238.305} C_VEL
LIN {X 0,Y 328.012,Z 862.474,A -85,B 0,C 180,E1 -30239.021,E2 -30239.021} C_VEL
LIN {X 0,Y 337.475,Z 842.407,A -85,B 0,C 180,E1 -30239.528,E2 -30239.528} C_VEL
LIN {X 0,Y 342.167,Z 831.157,A -85,B 0,C 180,E1 -30239.776,E2 -30239.776} C_VEL
LIN {X 0,Y 331.427,Z 855.703,A -85,B 0,C 180,E1 -30240.248,E2 -30240.248} C_VEL
LIN {X 0,Y 320.993,Z 875.773,A -85,B 0,C 180,E1 -30240.75,E2 -30240.75} C_VEL
LIN {X 0,Y 308.064,Z 897.368,A -85,B 0,C 180,E1 -30241.436,E2 -30241.436} C_VEL
LIN {X 0,Y 294.595,Z 916.731,A -85,B 0,C 180,E1 -30242.222,E2 -30242.222} C_VEL
LIN {X 0,Y 279.411,Z 936.123,A -85,B 0,C 180,E1 -30243.218,E2 -30243.218} C_VEL
LIN {X 0,Y 263.055,Z 954.248,A -85,B 0,C 180,E1 -30244.445,E2 -30244.445} C_VEL
LIN {X 0,Y 246.279,Z 970.915,A -85,B 0,C 180,E1 -30245.901,E2 -30245.901} C_VEL
LIN {X 0,Y 228.062,Z 986.796,A -85,B 0,C 180,E1 -30247.755,E2 -30247.755} C_VEL
LIN {X 0,Y 211.044,Z 1000.111,A -85,B 0,C 180,E1 -30249.821,E2 -30249.821} C_VEL
LIN {X 0,Y 203.239,Z 1005.726,A -85,B 0,C 180,E1 -30250.901,E2 -30250.901} C_VEL
LIN {X 0,Y 196.997,Z 1009.917,A -85,B 0,C 180,E1 -30251.511,E2 -30251.511} C_VEL
LIN {X 0,Y 178.783,Z 1020.494,A -85,B 0,C 180,E1 -30252.332,E2 -30252.332} C_VEL
LIN {X 0,Y 173.306,Z 1023.512,A -85,B 0,C 180,E1 -30253.036,E2 -30253.036} C_VEL
LIN {X 0,Y 153.846,Z 1034.141,A -85,B 0,C 180,E1 -30257.176,E2 -30257.176} C_VEL
LIN {X 0,Y 134.461,Z 1043.347,A -85,B 0,C 180,E1 -30262.764,E2 -30262.764} C_VEL
LIN {X 0,Y 117.433,Z 1050.636,A -85,B 0,C 180,E1 -30269.717,E2 -30269.717} C_VEL
LIN {X 0,Y 100.699,Z 1057.066,A -85,B 0,C 180,E1 -30280.197,E2 -30280.197} C_VEL
LIN {X 0,Y 89.454,Z 1061.207,A -85,B 0,C 180,E1 -30292.064,E2 -30292.064} C_VEL
LIN {X 0,Y 81.807,Z 1064.271,A -85,B 0,C 180,E1 -30308.489,E2 -30308.489} C_VEL
LIN {X 0,Y 80.039,Z 1065.385,A -85,B 0,C 180,E1 -30322.101,E2 -30322.101} C_VEL
LIN {X 0,Y 80.059,Z 1065.626,A -85,B 0,C 180,E1 -30330.715,E2 -30330.715} C_VEL
LIN {X 0,Y 80.188,Z 1065.246,A -85,B 0,C 180,E1 -30341.508,E2 -30341.508} C_VEL
LIN {X 0,Y 83.857,Z 1063.32,A -85,B 0,C 180,E1 -30357.711,E2 -30357.711} C_VEL
LIN {X 0,Y 91.677,Z 1060.327,A -85,B 0,C 180,E1 -30370.873,E2 -30370.873} C_VEL
LIN {X 0,Y 105.703,Z 1055.156,A -85,B 0,C 180,E1 -30383.518,E2 -30383.518} C_VEL
LIN {X 0,Y 121.136,Z 1048.989,A -85,B 0,C 180,E1 -30392.031,E2 -30392.031} C_VEL
LIN {X 0,Y 139.38,Z 1041.067,A -85,B 0,C 180,E1 -30398.842,E2 -30398.842} C_VEL
LIN {X 0,Y 159.094,Z 1031.198,A -85,B 0,C 180,E1 -30404.067,E2 -30404.067} C_VEL
LIN {X 0,Y 178.911,Z 1020.142,A -85,B 0,C 180,E1 -30407.967,E2 -30407.967} C_VEL
LIN {X 0,Y 199.058,Z 1007.19,A -85,B 0,C 180,E1 -30411.042,E2 -30411.042} C_VEL
LIN {X 0,Y 217.464,Z 993.976,A -85,B 0,C 180,E1 -30413.292,E2 -30413.292} C_VEL
LIN {X 0,Y 236.789,Z 978.161,A -85,B 0,C 180,E1 -30415.243,E2 -30415.243} C_VEL
LIN {X 0,Y 253.404,Z 962.914,A -85,B 0,C 180,E1 -30416.651,E2 -30416.651} C_VEL
LIN {X 0,Y 271.638,Z 943.905,A -85,B 0,C 180,E1 -30417.981,E2 -30417.981} C_VEL
LIN {X 0,Y 285.524,Z 927.54,A -85,B 0,C 180,E1 -30418.862,E2 -30418.862} C_VEL
LIN {X 0,Y 301.469,Z 906.22,A -85,B 0,C 180,E1 -30419.754,E2 -30419.754} C_VEL
LIN {X 0,Y 313.934,Z 887.012,A -85,B 0,C 180,E1 -30420.387,E2 -30420.387} C_VEL
LIN {X 0,Y 301.52,Z 906.028,A -85,B 0,C 180,E1 -30421.091,E2 -30421.091} C_VEL
LIN {X 0,Y 286.151,Z 926.499,A -85,B 0,C 180,E1 -30422.051,E2 -30422.051} C_VEL
LIN {X 0,Y 272.344,Z 942.703,A -85,B 0,C 180,E1 -30423.006,E2 -30423.006} C_VEL
LIN {X 0,Y 254.714,Z 961.062,A -85,B 0,C 180,E1 -30424.378,E2 -30424.378} C_VEL
LIN {X 0,Y 238.213,Z 976.13,A -85,B 0,C 180,E1 -30425.85,E2 -30425.85} C_VEL
LIN {X 0,Y 219.988,Z 991.07,A -85,B 0,C 180,E1 -30427.757,E2 -30427.757} C_VEL
LIN {X 0,Y 201.103,Z 1004.548,A -85,B 0,C 180,E1 -30430.115,E2 -30430.115} C_VEL
LIN {X 0,Y 182.622,Z 1016.354,A -85,B 0,C 180,E1 -30432.946,E2 -30432.946} C_VEL
LIN {X 0,Y 162.023,Z 1027.838,A -85,B 0,C 180,E1 -30436.953,E2 -30436.953} C_VEL
LIN {X 0,Y 143.843,Z 1036.793,A -85,B 0,C 180,E1 -30441.618,E2 -30441.618} C_VEL
LIN {X 0,Y 124.158,Z 1045.265,A -85,B 0,C 180,E1 -30448.62,E2 -30448.62} C_VEL
LIN {X 0,Y 108.538,Z 1051.238,A -85,B 0,C 180,E1 -30456.784,E2 -30456.784} C_VEL
LIN {X 0,Y 93.611,Z 1056.413,A -85,B 0,C 180,E1 -30469.341,E2 -30469.341} C_VEL
LIN {X 0,Y 85.259,Z 1059.209,A -85,B 0,C 180,E1 -30482.024,E2 -30482.024} C_VEL
LIN {X 0,Y 80.824,Z 1060.929,A -85,B 0,C 180,E1 -30497.134,E2 -30497.134} C_VEL
LIN {X 0,Y 80.074,Z 1061.351,A -85,B 0,C 180,E1 -30509.285,E2 -30509.285} C_VEL
LIN {X 0,Y 80.549,Z 1061.068,A -85,B 0,C 180,E1 -30520.732,E2 -30520.732} C_VEL
LIN {X 0,Y 84.641,Z 1059.475,A -85,B 0,C 180,E1 -30536.674,E2 -30536.674} C_VEL
LIN {X 0,Y 92.608,Z 1056.789,A -85,B 0,C 180,E1 -30549.571,E2 -30549.571} C_VEL
LIN {X 0,Y 105.945,Z 1052.316,A -85,B 0,C 180,E1 -30561.568,E2 -30561.568} C_VEL
LIN {X 0,Y 122.591,Z 1045.984,A -85,B 0,C 180,E1 -30570.778,E2 -30570.778} C_VEL
LIN {X 0,Y 140.693,Z 1038.417,A -85,B 0,C 180,E1 -30577.503,E2 -30577.503} C_VEL
LIN {X 0,Y 160.215,Z 1028.922,A -85,B 0,C 180,E1 -30582.721,E2 -30582.721} C_VEL
LIN {X 0,Y 179.842,Z 1018.215,A -85,B 0,C 180,E1 -30586.649,E2 -30586.649} C_VEL
LIN {X 0,Y 199.191,Z 1006.049,A -85,B 0,C 180,E1 -30589.696,E2 -30589.696} C_VEL
LIN {X 0,Y 217.096,Z 993.44,A -85,B 0,C 180,E1 -30591.988,E2 -30591.988} C_VEL
LIN {X 0,Y 236.254,Z 978.129,A -85,B 0,C 180,E1 -30594.035,E2 -30594.035} C_VEL
LIN {X 0,Y 251.766,Z 964.167,A -85,B 0,C 180,E1 -30595.451,E2 -30595.451} C_VEL
LIN {X 0,Y 268.741,Z 947.14,A -85,B 0,C 180,E1 -30596.801,E2 -30596.801} C_VEL
LIN {X 0,Y 284.161,Z 929.374,A -85,B 0,C 180,E1 -30597.894,E2 -30597.894} C_VEL
LIN {X 0,Y 298.532,Z 910.802,A -85,B 0,C 180,E1 -30598.808,E2 -30598.808} C_VEL
LIN {X 0,Y 312.474,Z 889.97,A -85,B 0,C 180,E1 -30599.607,E2 -30599.607} C_VEL
LIN {X 0,Y 313.343,Z 888.563,A -85,B 0,C 180,E1 -30599.655,E2 -30599.655} C_VEL
LIN {X 0,Y 299.973,Z 908.967,A -85,B 0,C 180,E1 -30600.339,E2 -30600.339} C_VEL
LIN {X 0,Y 285.03,Z 928.585,A -85,B 0,C 180,E1 -30601.179,E2 -30601.179} C_VEL
LIN {X 0,Y 270.347,Z 945.755,A -85,B 0,C 180,E1 -30602.12,E2 -30602.12} C_VEL
LIN {X 0,Y 252.427,Z 964.166,A -85,B 0,C 180,E1 -30603.438,E2 -30603.438} C_VEL
LIN {X 0,Y 236.794,Z 978.45,A -85,B 0,C 180,E1 -30604.768,E2 -30604.768} C_VEL
LIN {X 0,Y 217.47,Z 994.211,A -85,B 0,C 180,E1 -30606.718,E2 -30606.718} C_VEL
LIN {X 0,Y 199.167,Z 1007.327,A -85,B 0,C 180,E1 -30608.953,E2 -30608.953} C_VEL
LIN {X 0,Y 178.918,Z 1020.304,A -85,B 0,C 180,E1 -30612.041,E2 -30612.041} C_VEL
LIN {X 0,Y 173.306,Z 1023.512,A -85,B 0,C 180,E1 -30613.036,E2 -30613.036} C_VEL
LIN {X 0,Y 166.841,Z 1027.089,A -85,B 0,C 180,E1 -30613.892,E2 -30613.892} C_VEL
LIN {X 0,Y 147.911,Z 1035.817,A -85,B 0,C 180,E1 -30615.357,E2 -30615.357} C_VEL
LIN {X 0,Y 142.33,Z 1038.28,A -85,B 0,C 180,E1 -30616.379,E2 -30616.379} C_VEL
LIN {X 0,Y 121.889,Z 1047.164,A -85,B 0,C 180,E1 -30622.678,E2 -30622.678} C_VEL
LIN {X 0,Y 104.547,Z 1053.705,A -85,B 0,C 180,E1 -30630.597,E2 -30630.597} C_VEL
LIN {X 0,Y 88.901,Z 1059.157,A -85,B 0,C 180,E1 -30642.07,E2 -30642.07} C_VEL
LIN {X 0,Y 78.06,Z 1062.658,A -85,B 0,C 180,E1 -30656.578,E2 -30656.578} C_VEL
LIN {X 0,Y 73.017,Z 1064.566,A -85,B 0,C 180,E1 -30671.641,E2 -30671.641} C_VEL
LIN {X 0,Y 72.014,Z 1065.298,A -85,B 0,C 180,E1 -30685.221,E2 -30685.221} C_VEL
LIN {X 0,Y 72.026,Z 1065.341,A -85,B 0,C 180,E1 -30693.183,E2 -30693.183} C_VEL
LIN {X 0,Y 72.753,Z 1064.691,A -85,B 0,C 180,E1 -30706.774,E2 -30706.774} C_VEL
LIN {X 0,Y 77.357,Z 1062.862,A -85,B 0,C 180,E1 -30722.002,E2 -30722.002} C_VEL
LIN {X 0,Y 87.22,Z 1059.607,A -85,B 0,C 180,E1 -30736.238,E2 -30736.238} C_VEL
LIN {X 0,Y 103.108,Z 1054.149,A -85,B 0,C 180,E1 -30748.581,E2 -30748.581} C_VEL
LIN {X 0,Y 119.876,Z 1047.835,A -85,B 0,C 180,E1 -30756.564,E2 -30756.564} C_VEL
LIN {X 0,Y 140.949,Z 1038.795,A -85,B 0,C 180,E1 -30763.272,E2 -30763.272} C_VEL
LIN {X 0,Y 158.843,Z 1030.042,A -85,B 0,C 180,E1 -30767.342,E2 -30767.342} C_VEL
LIN {X 0,Y 180.19,Z 1018.213,A -85,B 0,C 180,E1 -30771.015,E2 -30771.015} C_VEL
LIN {X 0,Y 199.234,Z 1006.101,A -85,B 0,C 180,E1 -30773.562,E2 -30773.562} C_VEL
LIN {X 0,Y 219.58,Z 991.543,A -85,B 0,C 180,E1 -30775.746,E2 -30775.746} C_VEL
LIN {X 0,Y 237.677,Z 976.703,A -85,B 0,C 180,E1 -30777.348,E2 -30777.348} C_VEL
LIN {X 0,Y 256.036,Z 959.88,A -85,B 0,C 180,E1 -30778.711,E2 -30778.711} C_VEL
LIN {X 0,Y 272.971,Z 942.006,A -85,B 0,C 180,E1 -30779.797,E2 -30779.797} C_VEL
LIN {X 0,Y 284.978,Z 927.928,A -85,B 0,C 180,E1 -30780.488,E2 -30780.488} C_VEL
LIN {X 0,Y 270.55,Z 944.576,A -85,B 0,C 180,E1 -30781.398,E2 -30781.398} C_VEL
LIN {X 0,Y 252.251,Z 963.119,A -85,B 0,C 180,E1 -30782.697,E2 -30782.697} C_VEL
LIN {X 0,Y 235.566,Z 978.025,A -85,B 0,C 180,E1 -30784.064,E2 -30784.064} C_VEL
LIN {X 0,Y 215.17,Z 994.081,A -85,B 0,C 180,E1 -30786.039,E2 -30786.039} C_VEL
LIN {X 0,Y 197.924,Z 1006.023,A -85,B 0,C 180,E1 -30788.042,E2 -30788.042} C_VEL
LIN {X 0,Y 177.237,Z 1018.745,A -85,B 0,C 180,E1 -30791.001,E2 -30791.001} C_VEL
LIN {X 0,Y 158.017,Z 1028.961,A -85,B 0,C 180,E1 -30794.502,E2 -30794.502} C_VEL
LIN {X 0,Y 137.81,Z 1038.488,A -85,B 0,C 180,E1 -30799.401,E2 -30799.401} C_VEL
LIN {X 0,Y 118.852,Z 1046.078,A -85,B 0,C 180,E1 -30805.819,E2 -30805.819} C_VEL
LIN {X 0,Y 101.789,Z 1052.186,A -85,B 0,C 180,E1 -30814.397,E2 -30814.397} C_VEL
LIN {X 0,Y 87.037,Z 1056.786,A -85,B 0,C 180,E1 -30826.427,E2 -30826.427} C_VEL
LIN {X 0,Y 77.827,Z 1059.535,A -85,B 0,C 180,E1 -30839.931,E2 -30839.931} C_VEL
LIN {X 0,Y 72.758,Z 1061.254,A -85,B 0,C 180,E1 -30857.354,E2 -30857.354} C_VEL
LIN {X 0,Y 72.082,Z 1061.584,A -85,B 0,C 180,E1 -30870.001,E2 -30870.001} C_VEL
LIN {X 0,Y 72.753,Z 1061.263,A -85,B 0,C 180,E1 -30882.704,E2 -30882.704} C_VEL
LIN {X 0,Y 77.797,Z 1059.583,A -85,B 0,C 180,E1 -30900.084,E2 -30900.084} C_VEL
LIN {X 0,Y 86.988,Z 1056.853,A -85,B 0,C 180,E1 -30913.605,E2 -30913.605} C_VEL
LIN {X 0,Y 102.424,Z 1052.042,A -85,B 0,C 180,E1 -30926.078,E2 -30926.078} C_VEL
LIN {X 0,Y 118.795,Z 1046.202,A -85,B 0,C 180,E1 -30934.24,E2 -30934.24} C_VEL
LIN {X 0,Y 137.755,Z 1038.635,A -85,B 0,C 180,E1 -30940.666,E2 -30940.666} C_VEL
LIN {X 0,Y 157.968,Z 1029.14,A -85,B 0,C 180,E1 -30945.568,E2 -30945.568} C_VEL
LIN {X 0,Y 178.125,Z 1018.433,A -85,B 0,C 180,E1 -30949.219,E2 -30949.219} C_VEL
LIN {X 0,Y 197.889,Z 1006.265,A -85,B 0,C 180,E1 -30952.032,E2 -30952.032} C_VEL
LIN {X 0,Y 215.142,Z 994.349,A -85,B 0,C 180,E1 -30954.035,E2 -30954.035} C_VEL
LIN {X 0,Y 235.546,Z 978.344,A -85,B 0,C 180,E1 -30956.01,E2 -30956.01} C_VEL
LIN {X 0,Y 251.251,Z 964.382,A -85,B 0,C 180,E1 -30957.302,E2 -30957.302} C_VEL
LIN {X 0,Y 268.558,Z 947.19,A -85,B 0,C 180,E1 -30958.542,E2 -30958.542} C_VEL
LIN {X 0,Y 283.979,Z 929.586,A -85,B 0,C 180,E1 -30959.528,E2 -30959.528} C_VEL
LIN {X 0,Y 284.551,Z 928.892,A -85,B 0,C 180,E1 -30959.562,E2 -30959.562} C_VEL
LIN {X 0,Y 268.98,Z 946.871,A -85,B 0,C 180,E1 -30960.461,E2 -30960.461} C_VEL
LIN {X 0,Y 251.862,Z 964.145,A -85,B 0,C 180,E1 -30961.592,E2 -30961.592} C_VEL
LIN {X 0,Y 235.268,Z 979.086,A -85,B 0,C 180,E1 -30962.863,E2 -30962.863} C_VEL
LIN {X 0,Y 214.714,Z 995.409,A -85,B 0,C 180,E1 -30964.747,E2 -30964.747} C_VEL
LIN {X 0,Y 196.36,Z 1008.24,A -85,B 0,C 180,E1 -30966.799,E2 -30966.799} C_VEL
LIN {X 0,Y 174.279,Z 1021.81,A -85,B 0,C 180,E1 -30969.911,E2 -30969.911} C_VEL
LIN {X 0,Y 156.118,Z 1031.588,A -85,B 0,C 180,E1 -30973.215,E2 -30973.215} C_VEL
LIN {X 0,Y 142.33,Z 1038.28,A -85,B 0,C 180,E1 -30976.379,E2 -30976.379} C_VEL
LIN {X 0,Y 135.773,Z 1041.151,A -85,B 0,C 180,E1 -30977.644,E2 -30977.644} C_VEL
LIN {X 0,Y 116.99,Z 1047.804,A -85,B 0,C 180,E1 -30980.174,E2 -30980.174} C_VEL
LIN {X 0,Y 110.986,Z 1049.883,A -85,B 0,C 180,E1 -30981.874,E2 -30981.874} C_VEL
LIN {X 0,Y 90.959,Z 1056.609,A -85,B 0,C 180,E1 -30992.172,E2 -30992.172} C_VEL
LIN {X 0,Y 77.129,Z 1060.768,A -85,B 0,C 180,E1 -31004.519,E2 -31004.519} C_VEL
LIN {X 0,Y 66.892,Z 1063.836,A -85,B 0,C 180,E1 -31023.356,E2 -31023.356} C_VEL
LIN {X 0,Y 64.09,Z 1064.955,A -85,B 0,C 180,E1 -31040.118,E2 -31040.118} C_VEL
LIN {X 0,Y 64.059,Z 1065.199,A -85,B 0,C 180,E1 -31050.894,E2 -31050.894} C_VEL
LIN {X 0,Y 64.405,Z 1064.814,A -85,B 0,C 180,E1 -31064.382,E2 -31064.382} C_VEL
LIN {X 0,Y 69.766,Z 1062.882,A -85,B 0,C 180,E1 -31083.982,E2 -31083.982} C_VEL
LIN {X 0,Y 79.941,Z 1059.886,A -85,B 0,C 180,E1 -31098.63,E2 -31098.63} C_VEL
LIN {X 0,Y 96.774,Z 1054.712,A -85,B 0,C 180,E1 -31111.429,E2 -31111.429} C_VEL
LIN {X 0,Y 114.976,Z 1048.293,A -85,B 0,C 180,E1 -31119.643,E2 -31119.643} C_VEL
LIN {X 0,Y 136.08,Z 1039.81,A -85,B 0,C 180,E1 -31125.907,E2 -31125.907} C_VEL
LIN {X 0,Y 156.298,Z 1030.286,A -85,B 0,C 180,E1 -31130.125,E2 -31130.125} C_VEL
LIN {X 0,Y 177.164,Z 1019.152,A -85,B 0,C 180,E1 -31133.372,E2 -31133.372} C_VEL
LIN {X 0,Y 197.501,Z 1006.521,A -85,B 0,C 180,E1 -31135.828,E2 -31135.828} C_VEL
LIN {X 0,Y 217.147,Z 992.823,A -85,B 0,C 180,E1 -31137.723,E2 -31137.723} C_VEL
LIN {X 0,Y 236.682,Z 977.129,A -85,B 0,C 180,E1 -31139.274,E2 -31139.274} C_VEL
LIN {X 0,Y 253.978,Z 961.538,A -85,B 0,C 180,E1 -31140.423,E2 -31140.423} C_VEL
LIN {X 0,Y 256.274,Z 959.366,A -85,B 0,C 180,E1 -31140.563,E2 -31140.563} C_VEL
LIN {X 0,Y 238.097,Z 975.733,A -85,B 0,C 180,E1 -31141.849,E2 -31141.849} C_VEL
LIN {X 0,Y 220.345,Z 989.988,A -85,B 0,C 180,E1 -31143.321,E2 -31143.321} C_VEL
LIN {X 0,Y 199.849,Z 1004.362,A -85,B 0,C 180,E1 -31145.355,E2 -31145.355} C_VEL
LIN {X 0,Y 181.366,Z 1015.782,A -85,B 0,C 180,E1 -31147.603,E2 -31147.603} C_VEL
LIN {X 0,Y 158.944,Z 1027.828,A -85,B 0,C 180,E1 -31151.079,E2 -31151.079} C_VEL
LIN {X 0,Y 139.757,Z 1036.734,A -85,B 0,C 180,E1 -31155.016,E2 -31155.016} C_VEL
LIN {X 0,Y 117.308,Z 1045.659,A -85,B 0,C 180,E1 -31161.501,E2 -31161.501} C_VEL
LIN {X 0,Y 99.627,Z 1051.663,A -85,B 0,C 180,E1 -31169.173,E2 -31169.173} C_VEL
LIN {X 0,Y 81.901,Z 1056.85,A -85,B 0,C 180,E1 -31181.866,E2 -31181.866} C_VEL
LIN {X 0,Y 71.302,Z 1059.644,A -85,B 0,C 180,E1 -31195.881,E2 -31195.881} C_VEL
LIN {X 0,Y 65.213,Z 1061.359,A -85,B 0,C 180,E1 -31213.98,E2 -31213.98} C_VEL
LIN {X 0,Y 64.079,Z 1061.778,A -85,B 0,C 180,E1 -31229.107,E2 -31229.107} C_VEL
LIN {X 0,Y 64.69,Z 1061.517,A -85,B 0,C 180,E1 -31242.498,E2 -31242.498} C_VEL
LIN {X 0,Y 70.117,Z 1060.017,A -85,B 0,C 180,E1 -31261.846,E2 -31261.846} C_VEL
LIN {X 0,Y 80.677,Z 1057.224,A -85,B 0,C 180,E1 -31276.99,E2 -31276.99} C_VEL
LIN {X 0,Y 96.603,Z 1052.753,A -85,B 0,C 180,E1 -31289.216,E2 -31289.216} C_VEL
LIN {X 0,Y 115.46,Z 1046.421,A -85,B 0,C 180,E1 -31297.916,E2 -31297.916} C_VEL
LIN {X 0,Y 135.255,Z 1038.853,A -85,B 0,C 180,E1 -31303.956,E2 -31303.956} C_VEL
LIN {X 0,Y 156.123,Z 1029.357,A -85,B 0,C 180,E1 -31308.491,E2 -31308.491} C_VEL
LIN {X 0,Y 176.773,Z 1018.65,A -85,B 0,C 180,E1 -31311.835,E2 -31311.835} C_VEL
LIN {X 0,Y 197.722,Z 1005.962,A -85,B 0,C 180,E1 -31314.486,E2 -31314.486} C_VEL
LIN {X 0,Y 217.386,Z 992.486,A -85,B 0,C 180,E1 -31316.485,E2 -31316.485} C_VEL
LIN {X 0,Y 236.108,Z 977.722,A -85,B 0,C 180,E1 -31318.074,E2 -31318.074} C_VEL
LIN {X 0,Y 251.996,Z 963.678,A -85,B 0,C 180,E1 -31319.228,E2 -31319.228} C_VEL
LIN {X 0,Y 255.771,Z 960.199,A -85,B 0,C 180,E1 -31319.479,E2 -31319.479} C_VEL
LIN {X 0,Y 237.99,Z 976.311,A -85,B 0,C 180,E1 -31320.644,E2 -31320.644} C_VEL
LIN {X 0,Y 219.126,Z 991.59,A -85,B 0,C 180,E1 -31322.117,E2 -31322.117} C_VEL
LIN {X 0,Y 198.863,Z 1005.843,A -85,B 0,C 180,E1 -31324.037,E2 -31324.037} C_VEL
LIN {X 0,Y 179.089,Z 1018.179,A -85,B 0,C 180,E1 -31326.377,E2 -31326.377} C_VEL
LIN {X 0,Y 157.239,Z 1029.969,A -85,B 0,C 180,E1 -31329.716,E2 -31329.716} C_VEL
LIN {X 0,Y 137.889,Z 1039.12,A -85,B 0,C 180,E1 -31333.665,E2 -31333.665} C_VEL
LIN {X 0,Y 115.985,Z 1048.023,A -85,B 0,C 180,E1 -31340.003,E2 -31340.003} C_VEL
LIN {X 0,Y 110.986,Z 1049.883,A -85,B 0,C 180,E1 -31341.874,E2 -31341.874} C_VEL
LIN {X 0,Y 104.562,Z 1052.028,A -85,B 0,C 180,E1 -31343.902,E2 -31343.902} C_VEL
LIN {X 0,Y 85.633,Z 1056.862,A -85,B 0,C 180,E1 -31348.979,E2 -31348.979} C_VEL
LIN {X 0,Y 80.529,Z 1058.213,A -85,B 0,C 180,E1 -31351.783,E2 -31351.783} C_VEL
LIN {X 0,Y 65.484,Z 1062.101,A -85,B 0,C 180,E1 -31367.789,E2 -31367.789} C_VEL
LIN {X 0,Y 58.025,Z 1064.059,A -85,B 0,C 180,E1 -31385.57,E2 -31385.57} C_VEL
LIN {X 0,Y 56.026,Z 1064.844,A -85,B 0,C 180,E1 -31402.823,E2 -31402.823} C_VEL
LIN {X 0,Y 56.041,Z 1064.954,A -85,B 0,C 180,E1 -31412.35,E2 -31412.35} C_VEL
LIN {X 0,Y 57.021,Z 1064.402,A -85,B 0,C 180,E1 -31429.461,E2 -31429.461} C_VEL
LIN {X 0,Y 63.578,Z 1062.543,A -85,B 0,C 180,E1 -31448.981,E2 -31448.981} C_VEL
LIN {X 0,Y 76.063,Z 1059.332,A -85,B 0,C 180,E1 -31464.589,E2 -31464.589} C_VEL
LIN {X 0,Y 95.524,Z 1053.705,A -85,B 0,C 180,E1 -31477.091,E2 -31477.091} C_VEL
LIN {X 0,Y 114.294,Z 1047.39,A -85,B 0,C 180,E1 -31484.221,E2 -31484.221} C_VEL
LIN {X 0,Y 137.097,Z 1038.35,A -85,B 0,C 180,E1 -31489.927,E2 -31489.927} C_VEL
LIN {X 0,Y 156.799,Z 1029.233,A -85,B 0,C 180,E1 -31493.409,E2 -31493.409} C_VEL
LIN {X 0,Y 180.345,Z 1016.587,A -85,B 0,C 180,E1 -31496.503,E2 -31496.503} C_VEL
LIN {X 0,Y 199.054,Z 1005.013,A -85,B 0,C 180,E1 -31498.407,E2 -31498.407} C_VEL
LIN {X 0,Y 219.975,Z 990.32,A -85,B 0,C 180,E1 -31500.122,E2 -31500.122} C_VEL
LIN {X 0,Y 227.334,Z 984.605,A -85,B 0,C 180,E1 -31500.642,E2 -31500.642} C_VEL
LIN {X 0,Y 210.106,Z 997.294,A -85,B 0,C 180,E1 -31502.02,E2 -31502.02} C_VEL
LIN {X 0,Y 189.443,Z 1010.792,A -85,B 0,C 180,E1 -31504.015,E2 -31504.015} C_VEL
LIN {X 0,Y 169.057,Z 1022.23,A -85,B 0,C 180,E1 -31506.47,E2 -31506.47} C_VEL
LIN {X 0,Y 148.115,Z 1032.561,A -85,B 0,C 180,E1 -31509.734,E2 -31509.734} C_VEL
LIN {X 0,Y 126.875,Z 1041.355,A -85,B 0,C 180,E1 -31514.223,E2 -31514.223} C_VEL
LIN {X 0,Y 106.654,Z 1048.593,A -85,B 0,C 180,E1 -31520.364,E2 -31520.364} C_VEL
LIN {X 0,Y 87.319,Z 1054.303,A -85,B 0,C 180,E1 -31529.511,E2 -31529.511} C_VEL
LIN {X 0,Y 72.257,Z 1058.146,A -85,B 0,C 180,E1 -31541.648,E2 -31541.648} C_VEL
LIN {X 0,Y 60.143,Z 1060.907,A -85,B 0,C 180,E1 -31561.78,E2 -31561.78} C_VEL
LIN {X 0,Y 56.436,Z 1061.802,A -85,B 0,C 180,E1 -31579.796,E2 -31579.796} C_VEL
LIN {X 0,Y 56.098,Z 1061.957,A -85,B 0,C 180,E1 -31593.066,E2 -31593.066} C_VEL
LIN {X 0,Y 57.873,Z 1061.474,A -85,B 0,C 180,E1 -31610.216,E2 -31610.216} C_VEL
LIN {X 0,Y 65.162,Z 1059.8,A -85,B 0,C 180,E1 -31628.987,E2 -31628.987} C_VEL
LIN {X 0,Y 77.976,Z 1056.827,A -85,B 0,C 180,E1 -31643.888,E2 -31643.888} C_VEL
LIN {X 0,Y 96.653,Z 1051.735,A -85,B 0,C 180,E1 -31655.558,E2 -31655.558} C_VEL
LIN {X 0,Y 114.37,Z 1046.047,A -85,B 0,C 180,E1 -31662.354,E2 -31662.354} C_VEL
LIN {X 0,Y 136.897,Z 1037.51,A -85,B 0,C 180,E1 -31668.163,E2 -31668.163} C_VEL
LIN {X 0,Y 156.593,Z 1028.672,A -85,B 0,C 180,E1 -31671.78,E2 -31671.78} C_VEL
LIN {X 0,Y 178.704,Z 1017.227,A -85,B 0,C 180,E1 -31674.845,E2 -31674.845} C_VEL
LIN {X 0,Y 198.256,Z 1005.444,A -85,B 0,C 180,E1 -31676.971,E2 -31676.971} C_VEL
LIN {X 0,Y 218.031,Z 992.005,A -85,B 0,C 180,E1 -31678.72,E2 -31678.72} C_VEL
LIN {X 0,Y 226.86,Z 985.25,A -85,B 0,C 180,E1 -31679.401,E2 -31679.401} C_VEL
LIN {X 0,Y 208.995,Z 998.513,A -85,B 0,C 180,E1 -31680.745,E2 -31680.745} C_VEL
LIN {X 0,Y 186.213,Z 1013.313,A -85,B 0,C 180,E1 -31682.868,E2 -31682.868} C_VEL
LIN {X 0,Y 166.924,Z 1024.208,A -85,B 0,C 180,E1 -31685.155,E2 -31685.155} C_VEL
LIN {X 0,Y 143.629,Z 1035.619,A -85,B 0,C 180,E1 -31688.81,E2 -31688.81} C_VEL
LIN {X 0,Y 124.152,Z 1043.78,A -85,B 0,C 180,E1 -31693.033,E2 -31693.033} C_VEL
LIN {X 0,Y 102.172,Z 1051.696,A -85,B 0,C 180,E1 -31700.033,E2 -31700.033} C_VEL
LIN {X 0,Y 84.453,Z 1057.064,A -85,B 0,C 180,E1 -31709.041,E2 -31709.041} C_VEL
LIN {X 0,Y 80.529,Z 1058.213,A -85,B 0,C 180,E1 -31711.783,E2 -31711.783} C_VEL
LIN {X 0,Y 74.735,Z 1059.658,A -85,B 0,C 180,E1 -31715.448,E2 -31715.448} C_VEL
LIN {X 0,Y 57.527,Z 1062.536,A -85,B 0,C 180,E1 -31726.949,E2 -31726.949} C_VEL
LIN {X 0,Y 54.135,Z 1063.157,A -85,B 0,C 180,E1 -31732.152,E2 -31732.152} C_VEL
LIN {X 0,Y 48.336,Z 1064.496,A -85,B 0,C 180,E1 -31755.626,E2 -31755.626} C_VEL
LIN {X 0,Y 48.075,Z 1064.792,A -85,B 0,C 180,E1 -31769.999,E2 -31769.999} C_VEL
LIN {X 0,Y 48.565,Z 1064.435,A -85,B 0,C 180,E1 -31786.752,E2 -31786.752} C_VEL
LIN {X 0,Y 55.895,Z 1062.683,A -85,B 0,C 180,E1 -31811.443,E2 -31811.443} C_VEL
LIN {X 0,Y 69.415,Z 1059.611,A -85,B 0,C 180,E1 -31828.195,E2 -31828.195} C_VEL
LIN {X 0,Y 88.334,Z 1054.791,A -85,B 0,C 180,E1 -31839.968,E2 -31839.968} C_VEL
LIN {X 0,Y 108.65,Z 1048.41,A -85,B 0,C 180,E1 -31847.289,E2 -31847.289} C_VEL
LIN {X 0,Y 130.153,Z 1040.539,A -85,B 0,C 180,E1 -31852.318,E2 -31852.318} C_VEL
LIN {X 0,Y 152.366,Z 1030.773,A -85,B 0,C 180,E1 -31855.935,E2 -31855.935} C_VEL
LIN {X 0,Y 172.202,Z 1020.741,A -85,B 0,C 180,E1 -31858.336,E2 -31858.336} C_VEL
LIN {X 0,Y 194.984,Z 1007.362,A -85,B 0,C 180,E1 -31860.463,E2 -31860.463} C_VEL
LIN {X 0,Y 198.208,Z 1005.295,A -85,B 0,C 180,E1 -31860.721,E2 -31860.721} C_VEL
LIN {X 0,Y 178.485,Z 1017.053,A -85,B 0,C 180,E1 -31862.569,E2 -31862.569} C_VEL
LIN {X 0,Y 155.648,Z 1028.721,A -85,B 0,C 180,E1 -31865.302,E2 -31865.302} C_VEL
LIN {X 0,Y 135.474,Z 1037.573,A -85,B 0,C 180,E1 -31868.504,E2 -31868.504} C_VEL
LIN {X 0,Y 112.185,Z 1046.147,A -85,B 0,C 180,E1 -31873.713,E2 -31873.713} C_VEL
LIN {X 0,Y 92.737,Z 1052.103,A -85,B 0,C 180,E1 -31880.277,E2 -31880.277} C_VEL
LIN {X 0,Y 72.019,Z 1057.288,A -85,B 0,C 180,E1 -31892.125,E2 -31892.125} C_VEL
LIN {X 0,Y 58.539,Z 1060.079,A -85,B 0,C 180,E1 -31906.905,E2 -31906.905} C_VEL
LIN {X 0,Y 49.893,Z 1061.791,A -85,B 0,C 180,E1 -31928.856,E2 -31928.856} C_VEL
LIN {X 0,Y 48.09,Z 1062.183,A -85,B 0,C 180,E1 -31947.618,E2 -31947.618} C_VEL
LIN {X 0,Y 48.786,Z 1061.985,A -85,B 0,C 180,E1 -31964.239,E2 -31964.239} C_VEL
LIN {X 0,Y 55.496,Z 1060.776,A -85,B 0,C 180,E1 -31987.778,E2 -31987.778} C_VEL
LIN {X 0,Y 69.506,Z 1057.884,A -85,B 0,C 180,E1 -32005.872,E2 -32005.872} C_VEL
LIN {X 0,Y 86.821,Z 1053.803,A -85,B 0,C 180,E1 -32017.123,E2 -32017.123} C_VEL
LIN {X 0,Y 108.526,Z 1047.45,A -85,B 0,C 180,E1 -32025.332,E2 -32025.332} C_VEL
LIN {X 0,Y 127.891,Z 1040.675,A -85,B 0,C 180,E1 -32030.1,E2 -32030.1} C_VEL
LIN {X 0,Y 151.753,Z 1030.696,A -85,B 0,C 180,E1 -32034.229,E2 -32034.229} C_VEL
LIN {X 0,Y 171.262,Z 1021.115,A -85,B 0,C 180,E1 -32036.724,E2 -32036.724} C_VEL
LIN {X 0,Y 194.009,Z 1008.17,A -85,B 0,C 180,E1 -32038.994,E2 -32038.994} C_VEL
LIN {X 0,Y 197.777,Z 1005.796,A -85,B 0,C 180,E1 -32039.322,E2 -32039.322} C_VEL
LIN {X 0,Y 177.019,Z 1018.322,A -85,B 0,C 180,E1 -32041.176,E2 -32041.176} C_VEL
LIN {X 0,Y 155.152,Z 1029.601,A -85,B 0,C 180,E1 -32043.695,E2 -32043.695} C_VEL
LIN {X 0,Y 134.89,Z 1038.699,A -85,B 0,C 180,E1 -32046.811,E2 -32046.811} C_VEL
LIN {X 0,Y 111.406,Z 1047.582,A -85,B 0,C 180,E1 -32051.956,E2 -32051.956} C_VEL
LIN {X 0,Y 92.348,Z 1053.65,A -85,B 0,C 180,E1 -32058.3,E2 -32058.3} C_VEL
LIN {X 0,Y 70.865,Z 1059.331,A -85,B 0,C 180,E1 -32070.603,E2 -32070.603} C_VEL
LIN {X 0,Y 57.434,Z 1062.361,A -85,B 0,C 180,E1 -32085.862,E2 -32085.862} C_VEL
LIN {X 0,Y 54.135,Z 1063.157,A -85,B 0,C 180,E1 -32092.152,E2 -32092.152} C_VEL
LIN {X 0,Y 50.163,Z 1063.858,A -85,B 0,C 180,E1 -32100.168,E2 -32100.168} C_VEL
LIN {X 0,Y 44.066,Z 1064.478,A -85,B 0,C 180,E1 -32113.231,E2 -32113.231} C_VEL
LIN {X 0,Y 40.025,Z 1064.523,A -85,B 0,C 180,E1 -32133.46,E2 -32133.46} C_VEL
LIN {X 0,Y 42.329,Z 1063.894,A -85,B 0,C 180,E1 -32158.191,E2 -32158.191} C_VEL
LIN {X 0,Y 52.482,Z 1061.984,A -85,B 0,C 180,E1 -32181.363,E2 -32181.363} C_VEL
LIN {X 0,Y 69.622,Z 1058.527,A -85,B 0,C 180,E1 -32197.184,E2 -32197.184} C_VEL
LIN {X 0,Y 91.284,Z 1053,A -85,B 0,C 180,E1 -32207.125,E2 -32207.125} C_VEL
LIN {X 0,Y 111.892,Z 1046.634,A -85,B 0,C 180,E1 -32212.706,E2 -32212.706} C_VEL
LIN {X 0,Y 135.186,Z 1037.904,A -85,B 0,C 180,E1 -32216.869,E2 -32216.869} C_VEL
LIN {X 0,Y 155.988,Z 1028.685,A -85,B 0,C 180,E1 -32219.502,E2 -32219.502} C_VEL
LIN {X 0,Y 168.946,Z 1022.19,A -85,B 0,C 180,E1 -32220.8,E2 -32220.8} C_VEL
LIN {X 0,Y 148.202,Z 1032.1,A -85,B 0,C 180,E1 -32223.119,E2 -32223.119} C_VEL
LIN {X 0,Y 124.826,Z 1041.45,A -85,B 0,C 180,E1 -32226.654,E2 -32226.654} C_VEL
LIN {X 0,Y 104.587,Z 1048.242,A -85,B 0,C 180,E1 -32231.023,E2 -32231.023} C_VEL
LIN {X 0,Y 81.381,Z 1054.542,A -85,B 0,C 180,E1 -32238.905,E2 -32238.905} C_VEL
LIN {X 0,Y 64.114,Z 1058.276,A -85,B 0,C 180,E1 -32249.151,E2 -32249.151} C_VEL
LIN {X 0,Y 48.268,Z 1061.115,A -85,B 0,C 180,E1 -32268.481,E2 -32268.481} C_VEL
LIN {X 0,Y 40.874,Z 1062.211,A -85,B 0,C 180,E1 -32294.391,E2 -32294.391} C_VEL
LIN {X 0,Y 40.097,Z 1062.406,A -85,B 0,C 180,E1 -32312.86,E2 -32312.86} C_VEL
LIN {X 0,Y 42.748,Z 1061.969,A -85,B 0,C 180,E1 -32336.387,E2 -32336.387} C_VEL
LIN {X 0,Y 53.486,Z 1060.234,A -85,B 0,C 180,E1 -32360.04,E2 -32360.04} C_VEL
LIN {X 0,Y 69.592,Z 1057.263,A -85,B 0,C 180,E1 -32374.848,E2 -32374.848} C_VEL
LIN {X 0,Y 91.092,Z 1052.172,A -85,B 0,C 180,E1 -32385.008,E2 -32385.008} C_VEL
LIN {X 0,Y 110.502,Z 1046.484,A -85,B 0,C 180,E1 -32390.508,E2 -32390.508} C_VEL
LIN {X 0,Y 134.49,Z 1037.947,A -85,B 0,C 180,E1 -32395.039,E2 -32395.039} C_VEL
LIN {X 0,Y 155.098,Z 1029.108,A -85,B 0,C 180,E1 -32397.799,E2 -32397.799} C_VEL
LIN {X 0,Y 168.593,Z 1022.552,A -85,B 0,C 180,E1 -32399.242,E2 -32399.242} C_VEL
LIN {X 0,Y 146.047,Z 1033.501,A -85,B 0,C 180,E1 -32401.671,E2 -32401.671} C_VEL
LIN {X 0,Y 123.462,Z 1042.605,A -85,B 0,C 180,E1 -32405.027,E2 -32405.027} C_VEL
LIN {X 0,Y 101.477,Z 1050.155,A -85,B 0,C 180,E1 -32409.821,E2 -32409.821} C_VEL
LIN {X 0,Y 79.251,Z 1056.261,A -85,B 0,C 180,E1 -32417.626,E2 -32417.626} C_VEL
LIN {X 0,Y 60.388,Z 1060.54,A -85,B 0,C 180,E1 -32429.784,E2 -32429.784} C_VEL
LIN {X 0,Y 45.362,Z 1063.329,A -85,B 0,C 180,E1 -32451.888,E2 -32451.888} C_VEL
LIN {X 0,Y 40.299,Z 1064.334,A -85,B 0,C 180,E1 -32475.633,E2 -32475.633} C_VEL
LIN {X 0,Y 40.053,Z 1064.558,A -85,B 0,C 180,E1 -32491.429,E2 -32491.429} C_VEL
LIN {X 0,Y 40.025,Z 1064.523,A -85,B 0,C 180,E1 -32493.46,E2 -32493.46} C_VEL
LIN {X 0,Y 39.533,Z 1064.341,A -85,B 0,C 180,E1 -32502.994,E2 -32502.994} C_VEL
LIN {X 0,Y 38.573,Z 1063.966,A -85,B 0,C 180,E1 -32517.711,E2 -32517.711} C_VEL
LIN {X 0,Y 40.697,Z 1063.048,A -85,B 0,C 180,E1 -32537.148,E2 -32537.148} C_VEL
LIN {X 0,Y 43.664,Z 1062.466,A -85,B 0,C 180,E1 -32543.597,E2 -32543.597} C_VEL
LIN {X 0,Y 61.452,Z 1059.336,A -85,B 0,C 180,E1 -32560.683,E2 -32560.683} C_VEL
LIN {X 0,Y 83.17,Z 1054.589,A -85,B 0,C 180,E1 -32570.335,E2 -32570.335} C_VEL
LIN {X 0,Y 106.239,Z 1047.965,A -85,B 0,C 180,E1 -32576.054,E2 -32576.054} C_VEL
LIN {X 0,Y 128.987,Z 1040.094,A -85,B 0,C 180,E1 -32579.642,E2 -32579.642} C_VEL
LIN {X 0,Y 139.341,Z 1035.891,A -85,B 0,C 180,E1 -32580.888,E2 -32580.888} C_VEL
LIN {X 0,Y 118.245,Z 1043.747,A -85,B 0,C 180,E1 -32583.792,E2 -32583.792} C_VEL
LIN {X 0,Y 94.07,Z 1051.057,A -85,B 0,C 180,E1 -32588.696,E2 -32588.696} C_VEL
LIN {X 0,Y 73.646,Z 1055.962,A -85,B 0,C 180,E1 -32595.431,E2 -32595.431} C_VEL
LIN {X 0,Y 51.685,Z 1059.974,A -85,B 0,C 180,E1 -32609.477,E2 -32609.477} C_VEL
LIN {X 0,Y 37.967,Z 1061.839,A -85,B 0,C 180,E1 -32630.799,E2 -32630.799} C_VEL
LIN {X 0,Y 32.487,Z 1062.505,A -85,B 0,C 180,E1 -32657.56,E2 -32657.56} C_VEL
LIN {X 0,Y 32.143,Z 1062.596,A -85,B 0,C 180,E1 -32675.462,E2 -32675.462} C_VEL
LIN {X 0,Y 36.531,Z 1062.057,A -85,B 0,C 180,E1 -32705.087,E2 -32705.087} C_VEL
LIN {X 0,Y 49.39,Z 1060.343,A -85,B 0,C 180,E1 -32728.243,E2 -32728.243} C_VEL
LIN {X 0,Y 69.161,Z 1057.02,A -85,B 0,C 180,E1 -32742.592,E2 -32742.592} C_VEL
LIN {X 0,Y 91.208,Z 1051.896,A -85,B 0,C 180,E1 -32750.631,E2 -32750.631} C_VEL
LIN {X 0,Y 113.217,Z 1045.557,A -85,B 0,C 180,E1 -32755.441,E2 -32755.441} C_VEL
LIN {X 0,Y 137.01,Z 1036.971,A -85,B 0,C 180,E1 -32758.914,E2 -32758.914} C_VEL
LIN {X 0,Y 138.85,Z 1036.237,A -85,B 0,C 180,E1 -32759.175,E2 -32759.175} C_VEL
LIN {X 0,Y 116.076,Z 1044.91,A -85,B 0,C 180,E1 -32762.228,E2 -32762.228} C_VEL
LIN {X 0,Y 92.673,Z 1052.08,A -85,B 0,C 180,E1 -32766.957,E2 -32766.957} C_VEL
LIN {X 0,Y 71.168,Z 1057.438,A -85,B 0,C 180,E1 -32774.201,E2 -32774.201} C_VEL
LIN {X 0,Y 50.035,Z 1061.443,A -85,B 0,C 180,E1 -32788.441,E2 -32788.441} C_VEL
LIN {X 0,Y 36.668,Z 1063.48,A -85,B 0,C 180,E1 -32811.156,E2 -32811.156} C_VEL
LIN {X 0,Y 32.029,Z 1064.276,A -85,B 0,C 180,E1 -32842.825,E2 -32842.825} C_VEL
LIN {X 0,Y 32.02,Z 1064.294,A -85,B 0,C 180,E1 -32855.374,E2 -32855.374} C_VEL
LIN {X 0,Y 35.772,Z 1063.603,A -85,B 0,C 180,E1 -32885.941,E2 -32885.941} C_VEL
LIN {X 0,Y 43.664,Z 1062.466,A -85,B 0,C 180,E1 -32903.597,E2 -32903.597} C_VEL
LIN {X 0,Y 48.3,Z 1061.58,A -85,B 0,C 180,E1 -32911.293,E2 -32911.293} C_VEL
LIN {X 0,Y 62.053,Z 1058.764,A -85,B 0,C 180,E1 -32928.868,E2 -32928.868} C_VEL
LIN {X 0,Y 67.237,Z 1057.67,A -85,B 0,C 180,E1 -32931.588,E2 -32931.588} C_VEL
LIN {X 0,Y 90.056,Z 1052.294,A -85,B 0,C 180,E1 -32937.786,E2 -32937.786} C_VEL
LIN {X 0,Y 109.004,Z 1046.808,A -85,B 0,C 180,E1 -32941.014,E2 -32941.014} C_VEL
LIN {X 0,Y 87.313,Z 1052.763,A -85,B 0,C 180,E1 -32944.931,E2 -32944.931} C_VEL
LIN {X 0,Y 62.52,Z 1057.945,A -85,B 0,C 180,E1 -32952.69,E2 -32952.69} C_VEL
LIN {X 0,Y 43.983,Z 1060.733,A -85,B 0,C 180,E1 -32964.589,E2 -32964.589} C_VEL
LIN {X 0,Y 28.153,Z 1062.502,A -85,B 0,C 180,E1 -32992.861,E2 -32992.861} C_VEL
LIN {X 0,Y 24.095,Z 1062.846,A -85,B 0,C 180,E1 -33027.624,E2 -33027.624} C_VEL
LIN {X 0,Y 26.414,Z 1062.611,A -85,B 0,C 180,E1 -33059.481,E2 -33059.481} C_VEL
LIN {X 0,Y 41.524,Z 1061.101,A -85,B 0,C 180,E1 -33092.995,E2 -33092.995} C_VEL
LIN {X 0,Y 60.658,Z 1058.314,A -85,B 0,C 180,E1 -33106.548,E2 -33106.548} C_VEL
LIN {X 0,Y 83.414,Z 1053.845,A -85,B 0,C 180,E1 -33114.234,E2 -33114.234} C_VEL
LIN {X 0,Y 107.014,Z 1047.513,A -85,B 0,C 180,E1 -33118.773,E2 -33118.773} C_VEL
LIN {X 0,Y 108.693,Z 1047.016,A -85,B 0,C 180,E1 -33119.091,E2 -33119.091} C_VEL
LIN {X 0,Y 87.098,Z 1053.168,A -85,B 0,C 180,E1 -33122.839,E2 -33122.839} C_VEL
LIN {X 0,Y 62.031,Z 1058.671,A -85,B 0,C 180,E1 -33130.492,E2 -33130.492} C_VEL
LIN {X 0,Y 43.292,Z 1061.704,A -85,B 0,C 180,E1 -33142.5,E2 -33142.5} C_VEL
LIN {X 0,Y 27.027,Z 1063.738,A -85,B 0,C 180,E1 -33173.704,E2 -33173.704} C_VEL
LIN {X 0,Y 24.068,Z 1064.151,A -85,B 0,C 180,E1 -33209.998,E2 -33209.998} C_VEL
LIN {X 0,Y 27.026,Z 1063.73,A -85,B 0,C 180,E1 -33246.294,E2 -33246.294} C_VEL
LIN {X 0,Y 42.461,Z 1061.785,A -85,B 0,C 180,E1 -33276.689,E2 -33276.689} C_VEL
LIN {X 0,Y 62.029,Z 1058.615,A -85,B 0,C 180,E1 -33289.512,E2 -33289.512} C_VEL
LIN {X 0,Y 67.237,Z 1057.67,A -85,B 0,C 180,E1 -33291.588,E2 -33291.588} C_VEL
LIN {X 0,Y 67.858,Z 1057.477,A -85,B 0,C 180,E1 -33292.872,E2 -33292.872} C_VEL
LIN {X 0,Y 66.55,Z 1057.578,A -85,B 0,C 180,E1 -33295.622,E2 -33295.622} C_VEL
LIN {X 0,Y 62.52,Z 1058.088,A -85,B 0,C 180,E1 -33299.403,E2 -33299.403} C_VEL
LIN {X 0,Y 52.655,Z 1059.572,A -85,B 0,C 180,E1 -33305.968,E2 -33305.968} C_VEL
LIN {X 0,Y 43.552,Z 1060.694,A -85,B 0,C 180,E1 -33312.554,E2 -33312.554} C_VEL
LIN {X 0,Y 40.191,Z 1061.077,A -85,B 0,C 180,E1 -33314.975,E2 -33314.975} C_VEL
LIN {X 0,Y 20.969,Z 1062.78,A -85,B 0,C 180,E1 -33344.339,E2 -33344.339} C_VEL
LIN {X 0,Y 16.097,Z 1063.079,A -85,B 0,C 180,E1 -33390.003,E2 -33390.003} C_VEL
LIN {X 0,Y 20.958,Z 1062.789,A -85,B 0,C 180,E1 -33435.699,E2 -33435.699} C_VEL
LIN {X 0,Y 40.333,Z 1061.102,A -85,B 0,C 180,E1 -33465.21,E2 -33465.21} C_VEL
LIN {X 0,Y 60.263,Z 1058.378,A -85,B 0,C 180,E1 -33474.583,E2 -33474.583} C_VEL
LIN {X 0,Y 77.722,Z 1055.134,A -85,B 0,C 180,E1 -33478.938,E2 -33478.938} C_VEL
LIN {X 0,Y 56.162,Z 1059.284,A -85,B 0,C 180,E1 -33484.421,E2 -33484.421} C_VEL
LIN {X 0,Y 32.712,Z 1062.452,A -85,B 0,C 180,E1 -33498.634,E2 -33498.634} C_VEL
LIN {X 0,Y 17.807,Z 1063.686,A -85,B 0,C 180,E1 -33535.837,E2 -33535.837} C_VEL
LIN {X 0,Y 16.061,Z 1063.937,A -85,B 0,C 180,E1 -33569.997,E2 -33569.997} C_VEL
LIN {X 0,Y 21.672,Z 1063.461,A -85,B 0,C 180,E1 -33621.657,E2 -33621.657} C_VEL
LIN {X 0,Y 40.854,Z 1061.445,A -85,B 0,C 180,E1 -33648.231,E2 -33648.231} C_VEL
LIN {X 0,Y 62.053,Z 1058.227,A -85,B 0,C 180,E1 -33657.456,E2 -33657.456} C_VEL
LIN {X 0,Y 77.911,Z 1055.02,A -85,B 0,C 180,E1 -33661.102,E2 -33661.102} C_VEL
LIN {X 0,Y 56.39,Z 1058.932,A -85,B 0,C 180,E1 -33666.806,E2 -33666.806} C_VEL
LIN {X 0,Y 40.191,Z 1061.077,A -85,B 0,C 180,E1 -33674.975,E2 -33674.975} C_VEL
LIN {X 0,Y 32.984,Z 1061.848,A -85,B 0,C 180,E1 -33679.337,E2 -33679.337} C_VEL
LIN {X 0,Y 18.977,Z 1062.879,A -85,B 0,C 180,E1 -33688.211,E2 -33688.211} C_VEL
LIN {X 0,Y 9.62,Z 1063.18,A -85,B 0,C 180,E1 -33714.798,E2 -33714.798} C_VEL
LIN {X 0,Y 8.605,Z 1063.224,A -85,B 0,C 180,E1 -33727.428,E2 -33727.428} C_VEL
LIN {X 0,Y 9.773,Z 1063.177,A -85,B 0,C 180,E1 -33787.877,E2 -33787.877} C_VEL
LIN {X 0,Y 24.822,Z 1062.495,A -85,B 0,C 180,E1 -33828.38,E2 -33828.38} C_VEL
LIN {X 0,Y 44.377,Z 1060.74,A -85,B 0,C 180,E1 -33838.709,E2 -33838.709} C_VEL
LIN {X 0,Y 23.52,Z 1062.813,A -85,B 0,C 180,E1 -33849.791,E2 -33849.791} C_VEL
LIN {X 0,Y 8.29,Z 1063.657,A -85,B 0,C 180,E1 -33908.779,E2 -33908.779} C_VEL
LIN {X 0,Y 8.109,Z 1063.676,A -85,B 0,C 180,E1 -33944.27,E2 -33944.27} C_VEL
LIN {X 0,Y 22.404,Z 1062.875,A -85,B 0,C 180,E1 -34009.058,E2 -34009.058} C_VEL
LIN {X 0,Y 42.999,Z 1060.864,A -85,B 0,C 180,E1 -34020.852,E2 -34020.852} C_VEL
LIN {X 0,Y 44.282,Z 1060.707,A -85,B 0,C 180,E1 -34021.403,E2 -34021.403} C_VEL
LIN {X 0,Y 24.53,Z 1062.49,A -85,B 0,C 180,E1 -34031.971,E2 -34031.971} C_VEL
LIN {X 0,Y 9.78,Z 1063.169,A -85,B 0,C 180,E1 -34072.17,E2 -34072.17} C_VEL
LIN {X 0,Y 8.605,Z 1063.224,A -85,B 0,C 180,E1 -34087.428,E2 -34087.428} C_VEL
LIN {X 0,Y 7.08,Z 1063.302,A -85,B 0,C 180,E1 -34101.568,E2 -34101.568} C_VEL
LIN {X 0,Y 3.584,Z 1063.408,A -85,B 0,C 180,E1 -34132.639,E2 -34132.639} C_VEL
LIN {X 0,Y 1.669,Z 1063.473,A -85,B 0,C 180,E1 -34175.698,E2 -34175.698} C_VEL
LIN {X 0,Y 0.864,Z 1063.498,A -85,B 0,C 180,E1 -34195.858,E2 -34195.858} C_VEL
LIN {X 0,Y 0.862,Z 1063.49,A -85,B 0,C 180,E1 -34024.15,E2 -34024.15} C_VEL
LIN {X 0,Y 0.864,Z 1063.498,A -85,B 0,C 180,E1 -34195.858,E2 -34195.858} C_VEL
LIN {X 0,Y 2.884,Z 1065.498,A -85,B 0,C 180,E1 -34200.543,E2 -34200.543} C_VEL
LIN {X 0,Y 2.884,Z 1088.5,A -85,B 0,C 180,E1 -34200.543,E2 -34200.543} C_VEL
LIN {X 0,Y 2.884,Z 1088.5,A -85,B 0,C 180,E1 -34200.543,E2 -34200.543}

QRS_NEXT_CUT()

QRS_NEXT()
QRS_HOME()

END
